// Ошибка датчика давления не останавливает ГВС,
// но переводит подсистему в режим предупреждения (degraded mode).
IF fbPressValidator.VO_Error THEN
    GVL_STATE.G_DHW_Sensor_Fault := TRUE;
    GVL_STATE.G_DHW_Subsystem_Degraded := TRUE;
    VO_Status.Warning := TRUE;
    VO_Status.Error := FALSE;
    VO_Status.Error_ID := TO_WORD(GVL_CONFIG.ERR_DHW_PRESSURE_SENSOR_FAULT);
END_IF;

// 2. Логика поддержания температуры воды в бойлере (Нагрев)
// На этом этапе FB уже выполняется только на активном ПЛК.
    
// Термическая дезинфекция (Легионелла)
IF VI_Config.Anti_Legionella_Enabled
   AND (VI_Current_Day_Of_Week = VI_Config.Anti_Legionella_Day)
   AND (L_Current_TOD >= TOD#02:00)
   AND (L_Current_TOD <= TOD#04:00)
   AND NOT L_Legionella_Done_Today THEN
    L_Legionella_Active := TRUE;
ELSE
    L_Legionella_Active := FALSE;
END_IF;

L_Legionella_Timer(IN := L_Legionella_Active AND VO_Status.Temp >= 70.0, PT := T#30m, VI_System_Time_MS := VI_System_Time_MS);
IF L_Legionella_Timer.Q THEN
    L_Legionella_Active := FALSE; // Дезинфекция завершена
    L_Legionella_Done_Today := TRUE; // Повторно в те же сутки не запускать
END_IF;

// Двухпозиционное регулирование с гистерезисом
IF L_Legionella_Active THEN
    IF VO_Status.Temp < 70.0 THEN
        VO_Heating_Pump := TRUE;
    ELSIF VO_Status.Temp > 72.0 THEN
        VO_Heating_Pump := FALSE;
    END_IF;
ELSE
    IF VO_Status.Temp < (L_Target_Temp_Adjusted - VI_Config.Hysteresis) THEN
        VO_Heating_Pump := TRUE;
    ELSIF VO_Status.Temp > (L_Target_Temp_Adjusted + VI_Config.Hysteresis) THEN
        VO_Heating_Pump := FALSE;
    END_IF;
END_IF;

// 3. Управление циркуляционным насосом ГВС по расписанию
// Рециркуляция обеспечивает мгновенное наличие горячей воды у потребителя
VO_Circ_Pump := SEL(VI_Config.Circulation_Schedule_Enabled AND NOT (VI_Config.Night_Mode_Enabled AND (L_Current_TOD < VI_Config.Circulation_Start OR L_Current_TOD > VI_Config.Circulation_End)), FALSE, TRUE);

// Формирование статусных данных для визуализации.
// К этому моменту статус уже консистентен:
// - Error = критическая ошибка с остановкой ГВС
// - Warning = деградация без остановки
VO_Status.Heating_Pump_On := VO_Heating_Pump;
VO_Status.Circ_Pump_On := VO_Circ_Pump;

// >>> BULK_SYNC_ANCHOR: FB_DHW_Manager <<<
          
END_FUNCTION_BLOCK

FUNCTION_BLOCK FB_Safety_Manager
  VAR_INPUT
    VI_Gas_Alarm : BOOL;
    VI_Leak_Alarm : BOOL;
    VI_Smoke_Alarm : BOOL;
    VI_Reset : BOOL;
  END_VAR
  VAR_OUTPUT
    VO_Gas_Latched : BOOL;
    VO_Leak_Latched : BOOL;
    VO_Smoke_Latched : BOOL;
    VO_Emergency_Stop : BOOL;
  END_VAR
  VAR
    L_Any_Active : BOOL;
  END_VAR

            // Защёлкиваем аварии независимо друг от друга
IF VI_Gas_Alarm THEN
    VO_Gas_Latched := TRUE;
END_IF;

IF VI_Leak_Alarm THEN
    VO_Leak_Latched := TRUE;
END_IF;

IF VI_Smoke_Alarm THEN
    VO_Smoke_Latched := TRUE;
END_IF;

L_Any_Active := VI_Gas_Alarm OR VI_Leak_Alarm OR VI_Smoke_Alarm;

// Ручной сброс допустим только когда все входные аварийные сигналы уже исчезли
IF VI_Reset AND NOT L_Any_Active THEN
    VO_Gas_Latched := FALSE;
    VO_Leak_Latched := FALSE;
    VO_Smoke_Latched := FALSE;
END_IF;

// Агрегированный аварийный стоп = любая защёлкнутая safety-авария
VO_Emergency_Stop := VO_Gas_Latched OR VO_Leak_Latched OR VO_Smoke_Latched;

// >>> BULK_SYNC_ANCHOR: FB_Safety_Manager <<<
          
END_FUNCTION_BLOCK

FUNCTION_BLOCK FB_Calibration_Manager
  VAR_INPUT
    VI_Raw_Value : REAL;
    VI_Type : BYTE;
    VI_Calib_Record : ST_Sensor_Calibration_Record;
    VI_System_Time_MS : UDINT;
    VI_Start_Verification : BOOL;
  END_VAR
  VAR_OUTPUT
    VO_Calibrated_Value : REAL;
    VO_Verification_Active : BOOL;
    VO_Verification_Failed : BOOL;
    VO_Deviation_Percent : REAL;
  END_VAR
  VAR
    L_Verification_Timer : FB_System_Timer;
    L_Initial_Value : REAL;
  END_VAR

            // 1. Расчет калиброванного значения
CASE VI_Type OF
    1: VO_Calibrated_Value := VI_Raw_Value + VI_Calib_Record.offset;
    2, 3: VO_Calibrated_Value := (VI_Raw_Value * VI_Calib_Record.multiplier) + VI_Calib_Record.offset;
END_CASE;

// 2. Верификация через 1 час (ТЗ 9.5)
IF VI_Start_Verification AND NOT VO_Verification_Active THEN
    VO_Verification_Active := TRUE;
    L_Initial_Value := VO_Calibrated_Value;
END_IF;

L_Verification_Timer(IN := VO_Verification_Active, PT := T#1h, VI_System_Time_MS := VI_System_Time_MS);

IF L_Verification_Timer.Q THEN
    VO_Verification_Active := FALSE;
    
    // ТЗ 9.5: Отклонение ≤2.0% (норма) / >5.0% (ошибка)
    IF L_Initial_Value <> 0 THEN
        VO_Deviation_Percent := ABS(VO_Calibrated_Value - L_Initial_Value) / L_Initial_Value * 100.0;
    ELSE
        VO_Deviation_Percent := 0.0;
    END_IF;
    
    VO_Verification_Failed := (VO_Deviation_Percent > 5.0);
END_IF;
          
END_FUNCTION_BLOCK

FUNCTION_BLOCK FB_Persist_Pipeline
  VAR_INPUT
    VI_PersistStruct : ST_Persist;
    VI_System_Time_MS : UDINT;
    VI_IsActivePLC : BOOL;
  END_VAR
  VAR_OUTPUT
    VO_NVRAM_Cmd : BYTE;
    VO_NVRAM_Offset : UDINT;
    VO_NVRAM_Done : BOOL;
    VO_NVRAM_Err : BOOL;
    VO_NVRAM_ErrID : UDINT;
  END_VAR
  VAR_IN_OUT
    VIO_Apply_Settings : BOOL;
    VIO_Persist_Buffer : ARRAY[0..4] OF BYTE;
    VIO_Last_Written_Persist_Buffer : ARRAY[0..4] OF BYTE;
    VIO_Last_Persist_Write_MS : UDINT;
  END_VAR
  VAR
    fbNVRAMManager : FB_NVRAM_Manager;
    L_Persist_Buffer_Changed : BOOL;
  END_VAR

            // === SERIALIZE PERSIST STRUCT → BUFFER ===

// System Mode
VIO_Persist_Buffer[0] := TO_BYTE(TO_INT(VI_PersistStruct.System_Mode));

// Gas
IF VI_PersistStruct.Safety_Gas_Latched THEN
    VIO_Persist_Buffer[1] := BYTE#1;
ELSE
    VIO_Persist_Buffer[1] := BYTE#0;
END_IF;

// Smoke
IF VI_PersistStruct.Safety_Smoke_Latched THEN
    VIO_Persist_Buffer[2] := BYTE#1;
ELSE
    VIO_Persist_Buffer[2] := BYTE#0;
END_IF;

// Leak
IF VI_PersistStruct.Safety_Leak_Latched THEN
    VIO_Persist_Buffer[3] := BYTE#1;
ELSE
    VIO_Persist_Buffer[3] := BYTE#0;
END_IF;

// DHW Pump
IF VI_PersistStruct.DHW_Heating_Pump THEN
    VIO_Persist_Buffer[4] := BYTE#1;
ELSE
    VIO_Persist_Buffer[4] := BYTE#0;
END_IF;

// === END SERIALIZE ===

L_Persist_Buffer_Changed :=
    (VIO_Persist_Buffer[0] <> VIO_Last_Written_Persist_Buffer[0]) OR
    (VIO_Persist_Buffer[1] <> VIO_Last_Written_Persist_Buffer[1]) OR
    (VIO_Persist_Buffer[2] <> VIO_Last_Written_Persist_Buffer[2]) OR
    (VIO_Persist_Buffer[3] <> VIO_Last_Written_Persist_Buffer[3]) OR
    (VIO_Persist_Buffer[4] <> VIO_Last_Written_Persist_Buffer[4]);

VO_NVRAM_Cmd := 0;
VO_NVRAM_Offset := 0;

IF VIO_Apply_Settings THEN
    // explicit config apply requests a controlled write
    // keep flag set until successful write confirmation
    VO_NVRAM_Cmd := 1;

ELSIF L_Persist_Buffer_Changed THEN
    // controlled write: no more often than once per 60 seconds
    IF (VIO_Last_Persist_Write_MS = 0) OR
       ((VI_System_Time_MS - VIO_Last_Persist_Write_MS) >= 60000) THEN
        VO_NVRAM_Cmd := 1;
    END_IF;
END_IF;

fbNVRAMManager(
    VI_Command := VO_NVRAM_Cmd,
    VI_Offset := VO_NVRAM_Offset,
    VI_DataRef := VIO_Persist_Buffer[0],
    VI_DataSize := 5,
    VI_System_Time_MS := VI_System_Time_MS,
    VI_Operator_ID := 'SYSTEM',
    VI_IsActivePLC := VI_IsActivePLC,
    VI_TwoPersonConfirmation := FALSE,
    VO_Done => VO_NVRAM_Done,
    VO_Error => VO_NVRAM_Err,
    VO_ErrorID => VO_NVRAM_ErrID
);

IF (VO_NVRAM_Cmd = 1) AND VO_NVRAM_Done AND NOT VO_NVRAM_Err THEN
    VIO_Last_Written_Persist_Buffer[0] := VIO_Persist_Buffer[0];
    VIO_Last_Written_Persist_Buffer[1] := VIO_Persist_Buffer[1];
    VIO_Last_Written_Persist_Buffer[2] := VIO_Persist_Buffer[2];
    VIO_Last_Written_Persist_Buffer[3] := VIO_Persist_Buffer[3];
    VIO_Last_Written_Persist_Buffer[4] := VIO_Persist_Buffer[4];
    VIO_Last_Persist_Write_MS := VI_System_Time_MS;
    VIO_Apply_Settings := FALSE;
END_IF;
          
END_FUNCTION_BLOCK

FUNCTION_BLOCK FB_Boiler_Cascade_Manager
  VAR_INPUT
    VI_Enable : BOOL;
    VI_System_Time_MS : UDINT;
    VI_Boiler_Stop : BOOL;
    VI_DHW_Heating_Demand : BOOL;
    VI_DHW_Target_Temp : REAL;
    VI_Target_Supply_Temp : REAL;
    VI_Demand_Power : REAL;
    VI_Boiler_Flame_Status : ARRAY[1..GVL_CONSTANTS.C_MAX_BOILERS] OF BOOL;
    VI_Boiler_Error_Status : ARRAY[1..GVL_CONSTANTS.C_MAX_BOILERS] OF BOOL;
    VI_Boiler_OT_Online : ARRAY[1..GVL_CONSTANTS.C_MAX_BOILERS] OF BOOL;
    VI_Boiler_Modulation : ARRAY[1..GVL_CONSTANTS.C_MAX_BOILERS] OF REAL;
  END_VAR
  VAR_OUTPUT
    VO_Boiler_Enable : ARRAY[1..GVL_CONSTANTS.C_MAX_BOILERS] OF BOOL;
    VO_Boiler_Setpoint : ARRAY[1..GVL_CONSTANTS.C_MAX_BOILERS] OF REAL;
    VO_Lead_Boiler : BYTE;
  END_VAR
  VAR
    L_i : INT;
    L_Lead_Boiler : BYTE := 1;
    L_Last_Rotation_MS : UDINT := 0;
    L_Rotation_Initialized : BOOL := FALSE;
    L_Rotation_Period_MS : UDINT := 604800000;
    L_Lead_Available : BOOL;
    L_Reserve_Available : BOOL;
    L_Reserve_Boiler : BYTE;
    L_Start_Reserve : BOOL;
    L_Target_Setpoint : REAL;
    L_Flame_Miss_Timer : ARRAY[1..GVL_CONSTANTS.C_MAX_BOILERS] OF TON;
  END_VAR

            // Сброс выходов по умолчанию
FOR L_i := 1 TO GVL_CONSTANTS.C_MAX_BOILERS DO
    VO_Boiler_Enable[L_i] := FALSE;
    VO_Boiler_Setpoint[L_i] := 0.0;
END_FOR;

// Инициализация ротации
IF NOT L_Rotation_Initialized THEN
    L_Last_Rotation_MS := VI_System_Time_MS;
    L_Rotation_Initialized := TRUE;
END_IF;

// Принудительная остановка
IF VI_Boiler_Stop THEN
    VO_Lead_Boiler := L_Lead_Boiler;
    RETURN;
END_IF;

// Ротация строго каждые 168 часов
IF (VI_System_Time_MS - L_Last_Rotation_MS) >= L_Rotation_Period_MS THEN
    IF GVL_CONSTANTS.C_MAX_BOILERS > 1 THEN
        L_Lead_Boiler := 3 - L_Lead_Boiler;
    END_IF;
    L_Last_Rotation_MS := VI_System_Time_MS;
END_IF;

L_Reserve_Boiler := SEL(L_Lead_Boiler = 1, 1, 2);

L_Lead_Available :=
    VI_Boiler_OT_Online[L_Lead_Boiler] AND
    NOT VI_Boiler_Error_Status[L_Lead_Boiler];

L_Reserve_Available :=
    (GVL_CONSTANTS.C_MAX_BOILERS > 1) AND
    VI_Boiler_OT_Online[L_Reserve_Boiler] AND
    NOT VI_Boiler_Error_Status[L_Reserve_Boiler];

// Контроль "команда есть, пламени нет" для ведущего котла
L_Flame_Miss_Timer[L_Lead_Boiler](
    IN := VI_Enable AND L_Lead_Available AND NOT VI_DHW_Heating_Demand AND NOT VI_Boiler_Flame_Status[L_Lead_Boiler],
    PT := T#120s
);

IF L_Flame_Miss_Timer[L_Lead_Boiler].Q AND L_Reserve_Available THEN
    L_Lead_Boiler := L_Reserve_Boiler;
    L_Last_Rotation_MS := VI_System_Time_MS;
    L_Lead_Available :=
        VI_Boiler_OT_Online[L_Lead_Boiler] AND
        NOT VI_Boiler_Error_Status[L_Lead_Boiler];
    L_Reserve_Boiler := SEL(L_Lead_Boiler = 1, 1, 2);
    L_Reserve_Available :=
        (GVL_CONSTANTS.C_MAX_BOILERS > 1) AND
        VI_Boiler_OT_Online[L_Reserve_Boiler] AND
        NOT VI_Boiler_Error_Status[L_Reserve_Boiler];
END_IF;

// Нет запроса тепла
IF NOT VI_Enable THEN
    VO_Lead_Boiler := L_Lead_Boiler;
    RETURN;
END_IF;

// Целевая уставка
IF VI_DHW_Heating_Demand THEN
    L_Target_Setpoint := LIMIT(20.0, VI_DHW_Target_Temp + 15.0, 85.0);
ELSE
    L_Target_Setpoint := LIMIT(20.0, VI_Target_Supply_Temp + 5.0, 80.0);
END_IF;

// Выбор ведущего по доступности
IF NOT L_Lead_Available AND L_Reserve_Available THEN
    L_Lead_Boiler := L_Reserve_Boiler;
    L_Lead_Available := TRUE;
    L_Reserve_Boiler := SEL(L_Lead_Boiler = 1, 1, 2);
    L_Reserve_Available :=
        (GVL_CONSTANTS.C_MAX_BOILERS > 1) AND
        VI_Boiler_OT_Online[L_Reserve_Boiler] AND
        NOT VI_Boiler_Error_Status[L_Reserve_Boiler];
END_IF;

// Основной котёл
IF L_Lead_Available THEN
    VO_Boiler_Enable[L_Lead_Boiler] := TRUE;
    VO_Boiler_Setpoint[L_Lead_Boiler] := L_Target_Setpoint;
END_IF;

// Резервный котёл: >80% или отказ основного
L_Start_Reserve :=
    L_Reserve_Available AND
    (
        (VI_Demand_Power > 80.0) OR
        (NOT L_Lead_Available)
    );

IF L_Start_Reserve THEN
    VO_Boiler_Enable[L_Reserve_Boiler] := TRUE;
    VO_Boiler_Setpoint[L_Reserve_Boiler] := L_Target_Setpoint;
END_IF;

VO_Lead_Boiler := L_Lead_Boiler;
          
END_FUNCTION_BLOCK

FUNCTION_BLOCK FB_Watchdog
  VAR_INPUT
    VI_System_Time_MS : UDINT;
    VI_Timeout_MS : UDINT := 2000;
  END_VAR
  VAR_OUTPUT
    VO_Alive : BOOL;
    VO_Watchdog_Fault : BOOL;
    VO_Cycle_DT_MS : UDINT;
  END_VAR
  VAR
    L_Initialized : BOOL := FALSE;
    L_Last_Call_MS : UDINT := 0;
    L_DT_MS : UDINT := 0;
  END_VAR

            IF NOT L_Initialized THEN
    L_Initialized := TRUE;
    L_Last_Call_MS := VI_System_Time_MS;
    VO_Cycle_DT_MS := 0;
    VO_Watchdog_Fault := FALSE;
    VO_Alive := TRUE;
    RETURN;
END_IF;

// Measure real time gap between successive calls
L_DT_MS := (SEL(VI_System_Time_MS >= L_Last_Call_MS, VI_System_Time_MS - L_Last_Call_MS, (4294967295 - L_Last_Call_MS) + VI_System_Time_MS + 1));
VO_Cycle_DT_MS := L_DT_MS;

// Fault if the task/cycle resumed after an abnormal pause
VO_Watchdog_Fault := (L_DT_MS > VI_Timeout_MS);
VO_Alive := NOT VO_Watchdog_Fault;

// Store current timestamp for next cycle
L_Last_Call_MS := VI_System_Time_MS;
// >>> BULK_SYNC_ANCHOR: FB_Watchdog <<<
          
END_FUNCTION_BLOCK

FUNCTION_BLOCK FB_System_Health_Orchestrator
  VAR_OUTPUT
    VO_First_Fault_Active : BOOL;
    VO_First_Fault_Type : INT;
    VO_First_Fault_Source : INT;
    VO_System_Severity : E_System_Severity;
    VO_Root_Cause : E_System_Root_Cause;
    VO_Watchdog_Fault : BOOL;
  END_VAR
  VAR
    fbSafety : FB_Safety_Manager;
    fbWatchdog : FB_Watchdog;
    fbSystemHealth : FB_System_Health;
    fbStateManager : FB_State_Manager;
    fbHMIInterface : FB_HMI_Interface;
    fbFaultLogger : FB_Fault_Logger;
  END_VAR

            // ==============================================================================
// System health orchestrator helper
//
// Internal helper for PRG_System.
// Owns safety latch update, watchdog, system health aggregation,
// system mode calculation, HMI/fault publication, diagnostic exports,
// and human-readable mode/cause text projection.
// ==============================================================================



fbSafety(
    VI_Gas_Alarm := GVL_STATE.G_Safety_Gas_Alarm,
    VI_Leak_Alarm := GVL_STATE.G_Safety_Leak_Alarm,
    VI_Smoke_Alarm := GVL_STATE.G_Safety_Smoke_Alarm,
    VI_Reset := GVL_COMMAND.G_Reset_Errors,
    VO_Gas_Latched => GVL_STATE.G_Safety_Gas_Latched,
    VO_Leak_Latched => GVL_STATE.G_Safety_Leak_Latched,
    VO_Smoke_Latched => GVL_STATE.G_Safety_Smoke_Latched,
    VO_Emergency_Stop => GVL_STATE.G_Safety_Emergency_Stop
);

GVL_STATE.G_Freeze_Hardware_Degraded := GVL_STATUS.G_Diagnostics.Backup_Pump_Fault OR GVL_STATUS.G_Diagnostics.Electric_Heater_Fault;
GVL_STATE.G_Freeze_Hardware_Failed := GVL_STATUS.G_Diagnostics.Backup_Pump_Fault AND GVL_STATUS.G_Diagnostics.Electric_Heater_Fault;

fbWatchdog(
    VI_System_Time_MS := GVL_STATUS.G_System_Time_MS
);

fbSystemHealth(
    VI_Smoke_Detected := GVL_HEALTH_BRIDGE.G_Smoke_Detected OR GVL_STATE.G_Safety_Smoke_Latched,
    VI_Gas_Detected := GVL_HEALTH_BRIDGE.G_Gas_Detected OR GVL_STATE.G_Safety_Gas_Latched,
    VI_CO_Warning_Level := GVL_HEALTH_BRIDGE.G_CO_Warning_Level,
    VI_CO_Alarm_Level := GVL_HEALTH_BRIDGE.G_CO_Alarm_Level,
    VI_Leak_Detected := GVL_HEALTH_BRIDGE.G_Leak_Detected OR GVL_STATE.G_Safety_Leak_Latched,
    VI_Sensor_Fault := GVL_STATE.G_Heating_Sensor_Fault OR GVL_STATE.G_DHW_Sensor_Fault OR GVL_STATUS.G_Diagnostics.Manifold_Pressure_Fault_Active OR GVL_STATUS.G_Diagnostics.Manifold_Current_Fault_Active OR GVL_STATUS.G_Diagnostics.Manifold_Return_Temp_Fault_Active,
    VI_IO_Offline := GVL_STATE.G_Heating_IO_Fault OR GVL_STATE.G_DHW_IO_Fault OR GVL_STATE.G_Ventilation_IO_Fault OR GVL_STATE.G_Lighting_IO_Fault,
    VI_Comm_Fault := GVL_STATE.G_Access_Comm_Fault,
    VI_Watchdog_Fault := fbWatchdog.VO_Watchdog_Fault,
    VI_Subsystem_Fault := GVL_STATE.G_Heating_Subsystem_Degraded OR GVL_STATE.G_DHW_Subsystem_Degraded OR GVL_STATE.G_Ventilation_Subsystem_Degraded OR GVL_STATUS.G_Diagnostics.Manifold_Pressure_Fault_Active OR GVL_STATUS.G_Diagnostics.Manifold_Current_Fault_Active OR GVL_STATUS.G_Diagnostics.Manifold_Return_Temp_Fault_Active
);

fbStateManager(
    VI_System_Severity := fbSystemHealth.VO_System_Severity,
    VI_Root_Cause := fbSystemHealth.VO_Root_Cause,
    VI_Freeze_Risk := GVL_STATE.G_Safety_Freeze_Risk
);

fbHMIInterface(
    VI_Severity := fbSystemHealth.VO_System_Severity,
    VI_RootCause := fbSystemHealth.VO_Root_Cause,
    VI_Status_Msg := fbStateManager.VO_Status_Msg
);

fbFaultLogger(
    VI_Severity := fbSystemHealth.VO_System_Severity,
    VI_RootCause := fbSystemHealth.VO_Root_Cause,
    VI_Time_MS := GVL_STATUS.G_System_Time_MS
);

GVL_STATUS.G_System_Mode_Msg := fbStateManager.VO_Status_Msg;

GVL_STATUS.G_Diagnostics.Sensor_Fault :=
    GVL_STATE.G_Heating_Sensor_Fault OR
    GVL_STATE.G_DHW_Sensor_Fault OR
    GVL_STATUS.G_Diagnostics.Manifold_Pressure_Fault_Active OR
    GVL_STATUS.G_Diagnostics.Manifold_Current_Fault_Active OR
    GVL_STATUS.G_Diagnostics.Manifold_Return_Temp_Fault_Active;

GVL_STATUS.G_Diagnostics.IO_Offline :=
    GVL_STATE.G_Heating_IO_Fault OR
    GVL_STATE.G_DHW_IO_Fault OR
    GVL_STATE.G_Ventilation_IO_Fault OR
    GVL_STATE.G_Lighting_IO_Fault;

GVL_STATUS.G_Diagnostics.Subsystem_Degraded :=
    GVL_STATE.G_Heating_Subsystem_Degraded OR
    GVL_STATE.G_DHW_Subsystem_Degraded OR
    GVL_STATE.G_Ventilation_Subsystem_Degraded OR
    GVL_STATUS.G_Diagnostics.Manifold_Pressure_Fault_Active OR
    GVL_STATUS.G_Diagnostics.Manifold_Current_Fault_Active OR
    GVL_STATUS.G_Diagnostics.Manifold_Return_Temp_Fault_Active;

GVL_GATEWAY.G_Gateway_HMI_Status_Message := fbHMIInterface.VO_HMI_Status_Text;
IF fbFaultLogger.VO_Last_Event_Text <> '' THEN
    GVL_HEALTH_BRIDGE.G_Last_Fault_Event_Text := fbFaultLogger.VO_Last_Event_Text;
END_IF;

GVL_STATE.G_System_Mode := fbStateManager.VO_System_Mode;

CASE GVL_STATE.G_System_Mode OF
    E_System_Operating_Mode.MODE_SAFE_STOP:
        GVL_STATE.G_System_Mode_Text := 'SAFE_STOP';

    E_System_Operating_Mode.MODE_FREEZE_PROTECTION:
        GVL_STATE.G_System_Mode_Text := 'FREEZE_PROTECTION';

    E_System_Operating_Mode.MODE_DEGRADED:
        GVL_STATE.G_System_Mode_Text := 'DEGRADED';

    ELSE
        GVL_STATE.G_System_Mode_Text := 'NORMAL';
END_CASE;

CASE fbSystemHealth.VO_Root_Cause OF
    E_System_Root_Cause.ROOT_FIRE:
        GVL_STATUS.G_System_Mode_Cause := 'Пожар/дым';
    E_System_Root_Cause.ROOT_GAS_LEAK:
        GVL_STATUS.G_System_Mode_Cause := 'Утечка газа';
    E_System_Root_Cause.ROOT_CO_CRITICAL:
        GVL_STATUS.G_System_Mode_Cause := 'Критический CO';
    E_System_Root_Cause.ROOT_CO_WARNING:
        GVL_STATUS.G_System_Mode_Cause := 'Повышенный CO';
    E_System_Root_Cause.ROOT_WATER_LEAK:
        GVL_STATUS.G_System_Mode_Cause := 'Протечка воды';
    E_System_Root_Cause.ROOT_WATCHDOG_FAULT:
        GVL_STATUS.G_System_Mode_Cause := 'Ошибка watchdog';
    E_System_Root_Cause.ROOT_IO_OFFLINE:
        GVL_STATUS.G_System_Mode_Cause := 'Недоступен модуль IO';
    E_System_Root_Cause.ROOT_COMM_FAULT:
        GVL_STATUS.G_System_Mode_Cause := 'Ошибка связи';
    E_System_Root_Cause.ROOT_SENSOR_FAULT:
        GVL_STATUS.G_System_Mode_Cause := 'Ошибка датчика';
    E_System_Root_Cause.ROOT_SUBSYSTEM_FAULT:
        GVL_STATUS.G_System_Mode_Cause := 'Ошибка подсистемы';
    ELSE
        GVL_STATUS.G_System_Mode_Cause := 'Аварийные режимы отсутствуют';
END_CASE;

VO_First_Fault_Active := fbSystemHealth.VO_First_Fault_Active;
VO_First_Fault_Type := fbSystemHealth.VO_First_Fault_Type;
VO_First_Fault_Source := fbSystemHealth.VO_First_Fault_Source;
VO_System_Severity := fbSystemHealth.VO_System_Severity;
VO_Root_Cause := fbSystemHealth.VO_Root_Cause;
VO_Watchdog_Fault := fbWatchdog.VO_Watchdog_Fault;

GVL_STATUS.G_System_Mode_Msg := fbStateManager.VO_Status_Msg;

// >>> BULK_SYNC_ANCHOR: FB_System_Health_Orchestrator <<<
          
END_FUNCTION_BLOCK

FUNCTION_BLOCK FB_Diagnostics_Event_Manager
  VAR_INPUT
    VI_Code : UDINT;
    VI_Severity : INT;
    VI_Active : BOOL;
    VI_Timestamp : UDINT;
    VI_Source : INT;
  END_VAR
  VAR_IN_OUT
    VIO_Events : ARRAY[1..50] OF ST_Diagnostic_Event;
    VIO_Count : INT;
  END_VAR
  VAR
    L_i : INT;
    L_Found_Index : INT;
    L_Was_Active : BOOL;
  END_VAR

            L_Found_Index := 0;
L_Was_Active := FALSE;

FOR L_i := 1 TO VIO_Count DO
    IF (VIO_Events[L_i].Code = VI_Code) AND (VIO_Events[L_i].Source = VI_Source) THEN
        L_Found_Index := L_i;
        L_Was_Active := VIO_Events[L_i].Active;
    END_IF;
END_FOR;

IF VI_Active THEN
    IF L_Found_Index = 0 THEN
        IF VIO_Count < 50 THEN
            VIO_Count := VIO_Count + 1;
            VIO_Events[VIO_Count].Code := VI_Code;
            VIO_Events[VIO_Count].Severity := VI_Severity;
            VIO_Events[VIO_Count].Active := TRUE;
            VIO_Events[VIO_Count].Timestamp := VI_Timestamp;
            VIO_Events[VIO_Count].Source := VI_Source;
        END_IF;
    ELSE
        VIO_Events[L_Found_Index].Severity := VI_Severity;
        IF NOT L_Was_Active THEN
            VIO_Events[L_Found_Index].Timestamp := VI_Timestamp;
        END_IF;
        VIO_Events[L_Found_Index].Active := TRUE;
    END_IF;
ELSE
    IF L_Found_Index > 0 THEN
        VIO_Events[L_Found_Index].Active := FALSE;
    END_IF;
END_IF;
          
END_FUNCTION_BLOCK

PROGRAM PRG_Command_Arbitration
  VAR
    L_i : INT;
  END_VAR

            // Reset shadow operational commands before each arbitration cycle
GVL_COMMAND_SHADOW.G_Gas_Valve_Close := FALSE;
GVL_COMMAND_SHADOW.G_Boiler_Stop := FALSE;
GVL_COMMAND_SHADOW.G_Supply_100_Req := FALSE;
GVL_COMMAND_SHADOW.G_Supply_80_Req := FALSE;
GVL_COMMAND_SHADOW.G_Vent_PV3_Boost := FALSE;
GVL_COMMAND_SHADOW.G_Exhaust_100_Req := FALSE;
GVL_COMMAND_SHADOW.G_Vent_Stop := FALSE;

GVL_COMMAND_SHADOW.G_Close_Valve_35 := FALSE;
GVL_COMMAND_SHADOW.G_Close_Valve_36 := FALSE;

GVL_COMMAND_SHADOW.G_Lock_1_Open := FALSE;
GVL_COMMAND_SHADOW.G_Lock_1_Close := FALSE;
GVL_COMMAND_SHADOW.G_Lock_2_Open := FALSE;
GVL_COMMAND_SHADOW.G_Lock_2_Close := FALSE;
GVL_COMMAND_SHADOW.G_Gate_Open := FALSE;
GVL_COMMAND_SHADOW.G_Wicket_Open := FALSE;

// User intent pass-through into the shadow operational layer
GVL_COMMAND_SHADOW.G_Gate_Open := GVL_INTENT_USER.I_Gate_Open_Request;
GVL_COMMAND_SHADOW.G_Wicket_Open := GVL_INTENT_USER.I_Wicket_Open_Request;
GVL_COMMAND_SHADOW.G_Lock_1_Open := GVL_INTENT_USER.I_Lock_1_Open_Request;
GVL_COMMAND_SHADOW.G_Lock_1_Close := GVL_INTENT_USER.I_Lock_1_Close_Request;
GVL_COMMAND_SHADOW.G_Lock_2_Open := GVL_INTENT_USER.I_Lock_2_Open_Request;
GVL_COMMAND_SHADOW.G_Lock_2_Close := GVL_INTENT_USER.I_Lock_2_Close_Request;

// Safety and system arbitration into the shadow operational layer
IF GVL_INTENT_SAFETY.I_Fire_Alarm_Active THEN
    GVL_COMMAND_SHADOW.G_Boiler_Stop := TRUE;
    GVL_COMMAND_SHADOW.G_Vent_Stop := TRUE;
    GVL_COMMAND_SHADOW.G_Lock_1_Open := TRUE;
    GVL_COMMAND_SHADOW.G_Lock_2_Open := TRUE;
END_IF;

IF GVL_INTENT_SAFETY.I_Gas_Close_Required THEN
    GVL_COMMAND_SHADOW.G_Gas_Valve_Close := TRUE;
    GVL_COMMAND_SHADOW.G_Boiler_Stop := TRUE;
END_IF;

IF GVL_INTENT_SAFETY.I_Vent_Force_PV3_Boost THEN
    GVL_COMMAND_SHADOW.G_Vent_PV3_Boost := TRUE;
END_IF;

IF GVL_INTENT_SAFETY.I_Vent_Force_Supply_100 THEN
    GVL_COMMAND_SHADOW.G_Supply_100_Req := TRUE;
END_IF;

IF GVL_INTENT_SAFETY.I_Vent_Force_Supply_80 THEN
    GVL_COMMAND_SHADOW.G_Supply_80_Req := TRUE;
END_IF;

IF GVL_INTENT_SAFETY.I_Vent_Stop_Required THEN
    GVL_COMMAND_SHADOW.G_Vent_Stop := TRUE;
END_IF;

IF GVL_INTENT_SYSTEM.I_Mode_Degraded_Active THEN
    GVL_COMMAND_SHADOW.G_Supply_80_Req := TRUE;
END_IF;

IF GVL_INTENT_SAFETY.I_Water_Main_Close_Required THEN
    GVL_COMMAND_SHADOW.G_Close_Valve_35 := TRUE;
    GVL_COMMAND_SHADOW.G_Close_Valve_36 := TRUE;
END_IF;

FOR L_i := 1 TO 32 DO
    IF GVL_INTENT_SAFETY.I_Water_Zone_Close_Required[L_i] THEN
        ;
    END_IF;
END_FOR;
          
END_PROGRAM

PROGRAM PRG_PLC_A

            // Вызов основной программы
PRG_System();
// >>> BULK_SYNC_ANCHOR: PRG_PLC_A <<<
          
END_PROGRAM

PROGRAM PRG_Policy

            // ============================================================
// SCENARIO POLICY OWNER
// ============================================================

// 1. Base priority resolution
IF GVL_STATE.G_System_Mode = E_System_Operating_Mode.MODE_SAFE_STOP THEN
    GVL_POLICY.G_Scenario_Intent := E_SCENARIO_TYPE.SCENARIO_NONE;
    GVL_POLICY.G_Scenario_Source := SRC_SAFETY;

ELSIF GVL_POLICY.G_Scenario_Request_Operator <> E_SCENARIO_TYPE.SCENARIO_NONE THEN
    GVL_POLICY.G_Scenario_Intent := GVL_POLICY.G_Scenario_Request_Operator;
    GVL_POLICY.G_Scenario_Source := SRC_OPERATOR;

ELSIF GVL_POLICY.G_Scenario_Request_Gateway <> E_SCENARIO_TYPE.SCENARIO_NONE THEN
    GVL_POLICY.G_Scenario_Intent := GVL_POLICY.G_Scenario_Request_Gateway;
    GVL_POLICY.G_Scenario_Source := SRC_GATEWAY;

ELSIF GVL_POLICY.G_Scenario_Request_Rule <> E_SCENARIO_TYPE.SCENARIO_NONE THEN
    GVL_POLICY.G_Scenario_Intent := GVL_POLICY.G_Scenario_Request_Rule;
    GVL_POLICY.G_Scenario_Source := SRC_RULE;

ELSE
    GVL_POLICY.G_Scenario_Intent := GVL_STATUS.G_Current_Scenario;
    GVL_POLICY.G_Scenario_Source := SRC_NONE;
END_IF;

// 2. Fail-safe clamp
CASE GVL_STATE.G_System_Mode OF
    E_System_Operating_Mode.MODE_SAFE_STOP:
        GVL_POLICY.G_Scenario_Intent := E_SCENARIO_TYPE.SCENARIO_NONE;
        GVL_POLICY.G_Scenario_Source := SRC_SAFETY;

    E_System_Operating_Mode.MODE_FREEZE_PROTECTION:
        GVL_POLICY.G_Scenario_Intent := E_SCENARIO_TYPE.SCENARIO_NONE;
        GVL_POLICY.G_Scenario_Source := SRC_POLICY;

    E_System_Operating_Mode.MODE_DEGRADED:
        CASE GVL_POLICY.G_Scenario_Intent OF
            E_SCENARIO_TYPE.SCENARIO_NONE,
            E_SCENARIO_TYPE.SCENARIO_PRESENCE,
            E_SCENARIO_TYPE.SCENARIO_AWAY,
            E_SCENARIO_TYPE.SCENARIO_SLEEP:
                ;
        ELSE
            GVL_POLICY.G_Scenario_Intent := E_SCENARIO_TYPE.SCENARIO_NONE;
            GVL_POLICY.G_Scenario_Source := SRC_POLICY;
        END_CASE;
END_CASE;

// 3. Context automation
IF GVL_STATE.G_System_Mode = E_System_Operating_Mode.MODE_NORMAL THEN
    IF GVL_ALARM.G_Security_Armed AND
       (GVL_POLICY.G_Scenario_Request_Operator = E_SCENARIO_TYPE.SCENARIO_NONE) AND
       (GVL_POLICY.G_Scenario_Request_Gateway = E_SCENARIO_TYPE.SCENARIO_NONE) AND
       (GVL_POLICY.G_Scenario_Request_Rule = E_SCENARIO_TYPE.SCENARIO_NONE) AND
       (GVL_POLICY.G_Scenario_Intent <> E_SCENARIO_TYPE.SCENARIO_AWAY) THEN
        GVL_POLICY.G_Scenario_Intent := E_SCENARIO_TYPE.SCENARIO_AWAY;
        GVL_POLICY.G_Scenario_Source := SRC_POLICY;
    END_IF;
END_IF;

// 4. Degraded adaptation
IF GVL_STATE.G_System_Mode = E_System_Operating_Mode.MODE_DEGRADED THEN
    IF (GVL_POLICY.G_Scenario_Request_Operator = E_SCENARIO_TYPE.SCENARIO_NONE) AND
       (GVL_POLICY.G_Scenario_Request_Gateway = E_SCENARIO_TYPE.SCENARIO_NONE) AND
       (GVL_POLICY.G_Scenario_Request_Rule = E_SCENARIO_TYPE.SCENARIO_NONE) THEN

        IF GVL_ALARM.G_Security_Armed THEN
            GVL_POLICY.G_Scenario_Intent := E_SCENARIO_TYPE.SCENARIO_AWAY;
            GVL_POLICY.G_Scenario_Source := SRC_POLICY;

        ELSIF GVL_POLICY.G_Scenario_Intent = E_SCENARIO_TYPE.SCENARIO_PRESENCE THEN
            GVL_POLICY.G_Scenario_Intent := E_SCENARIO_TYPE.SCENARIO_SLEEP;
            GVL_POLICY.G_Scenario_Source := SRC_POLICY;
        END_IF;
    END_IF;
END_IF;

// 5. Heating bridge
GVL_STATE.G_Preheat_Request := GVL_POLICY.G_Rule_Preheat_Request;
GVL_STATE.G_Freeze_Request :=
    (GVL_STATE.G_System_Mode = E_System_Operating_Mode.MODE_FREEZE_PROTECTION);
          
END_PROGRAM

PROGRAM PRG_Safety
  VAR
    fbWaterLeakageManager : FB_Water_Leakage_Manager;
    fbGasSmokeManager : FB_Gas_Smoke_Manager;
    fbSafetyWorkflow : FB_Safety_Workflow_Manager;
    fbOwnership : FB_Ownership_Watchdog;
    L_i : INT;
  END_VAR

            // ========================================
// SAFETY_INTENT_RESET_INIT
// ========================================
GVL_INTENT_SAFETY.I_Source_Valid := TRUE;
GVL_INTENT_SAFETY.I_Last_Update_MS := GVL_STATUS.G_System_Time_MS;
GVL_INTENT_SAFETY.I_Fire_Alarm_Active := FALSE;
GVL_INTENT_SAFETY.I_Gas_Alarm_Active := FALSE;
GVL_INTENT_SAFETY.I_Leak_Alarm_Active := FALSE;
GVL_INTENT_SAFETY.I_CO_Warning_Active := FALSE;
GVL_INTENT_SAFETY.I_System_Safe_Stop_Required := FALSE;
GVL_INTENT_SAFETY.I_Freeze_Protection_Required := FALSE;
GVL_INTENT_SAFETY.I_Evacuation_Mode_Active := FALSE;
GVL_INTENT_SAFETY.I_Gas_Close_Required := FALSE;
GVL_INTENT_SAFETY.I_Boiler_Stop_Required := FALSE;
GVL_INTENT_SAFETY.I_Vent_Stop_Required := FALSE;
GVL_INTENT_SAFETY.I_Vent_Force_PV3_Boost := FALSE;
GVL_INTENT_SAFETY.I_Vent_Force_Supply_100 := FALSE;
GVL_INTENT_SAFETY.I_Vent_Force_Supply_80 := FALSE;
GVL_INTENT_SAFETY.I_Vent_Force_Exhaust_100 := FALSE;
GVL_INTENT_SAFETY.I_Water_Main_Close_Required := FALSE;
GVL_INTENT_SAFETY.I_Water_Selective_Recovery_Allowed := FALSE;
GVL_INTENT_SAFETY.I_Water_Recovery_Target_Zone := 0;
GVL_INTENT_SAFETY.I_Lock_1_Force_Open := FALSE;
GVL_INTENT_SAFETY.I_Lock_1_Force_Close_Block := FALSE;
GVL_INTENT_SAFETY.I_Lock_2_Force_Open := FALSE;
GVL_INTENT_SAFETY.I_Lock_2_Force_Close_Block := FALSE;

// ========================================
// SAFETY_WORKFLOW_FB
// ========================================
fbSafetyWorkflow(
    VI_System_Time_MS := GVL_STATUS.G_System_Time_MS,
    VI_Water_Selective_Recover := GVL_INTENT_USER.I_Water_Selective_Recover,
    VI_Gas_Selective_Recover := GVL_INTENT_USER.I_Gas_Selective_Recover,
    VI_Water_Valve_Test_Open := GVL_INTENT_USER.I_Water_Valve_Test_Open,
    VI_Water_Valve_Test_Close := GVL_INTENT_USER.I_Water_Valve_Test_Close,
    VI_Water_Valve_Test_Confirm := GVL_INTENT_USER.I_Water_Valve_Test_Confirm,
    VI_Gas_Valve_Test_Open := GVL_INTENT_USER.I_Gas_Valve_Test_Open,
    VI_Gas_Valve_Test_Close := GVL_INTENT_USER.I_Gas_Valve_Test_Close,
    VI_Gas_Valve_Test_Confirm := GVL_INTENT_USER.I_Gas_Valve_Test_Confirm
);

IF fbSafetyWorkflow.VO_Water_Test_Timeout_Close_Required THEN
    GVL_INTENT_SAFETY.I_Water_Main_Close_Required := TRUE;
END_IF;

IF fbSafetyWorkflow.VO_Gas_Test_Timeout_Close_Required THEN
    GVL_INTENT_SAFETY.I_Gas_Close_Required := TRUE;
END_IF;

// ========================================
// SAFETY_DETECTORS_AND_HEALTH_PROJECTION
// ========================================
fbWaterLeakageManager(
    VI_System_Time_MS := GVL_STATUS.G_System_Time_MS,
    VI_IsActivePLC := GVL_STATUS.G_Is_Active_PLC,
    VI_Sensors := GVL_STATE.G_Water_Sensors,
    VI_Config := GVL_CONFIG.G_HMI_Flood_Config,
    VO_Status_Msg => GVL_STATUS.G_Flood_Status_Msg,
    VO_Leak_Detected => GVL_HEALTH_BRIDGE.G_Leak_Detected,
    VO_Leak_Warning_Level => GVL_HEALTH_BRIDGE.G_Leak_Warning_Level
);
GVL_INTENT_SAFETY.I_Leak_Alarm_Active := GVL_HEALTH_BRIDGE.G_Leak_Detected;

fbGasSmokeManager(
    VI_System_Time_MS := GVL_STATUS.G_System_Time_MS,
    VI_IsActivePLC := GVL_STATUS.G_Is_Active_PLC,
    VI_Methane_LEL := GVL_Safety_Selector.G_Methane_Effective_Array,
    VI_CO_PPM := GVL_Safety_Selector.G_CO_Effective_Array,
    VI_Smoke_Sensors := GVL_Safety_Selector.G_Smoke_Effective_Array,
    VI_Mute_Request := GVL_CONFIG.G_HMI_Mute_Alarm,
    VO_Smoke_Detected => GVL_HEALTH_BRIDGE.G_Smoke_Detected,
    VO_Gas_Detected => GVL_HEALTH_BRIDGE.G_Gas_Detected,
    VO_CO_Warning_Level => GVL_HEALTH_BRIDGE.G_CO_Warning_Level,
    VO_CO_Alarm_Level => GVL_HEALTH_BRIDGE.G_CO_Alarm_Level,
    VO_Status_Msg => GVL_STATUS.G_Gas_Status_Msg
);
GVL_INTENT_SAFETY.I_Fire_Alarm_Active := GVL_HEALTH_BRIDGE.G_Smoke_Detected;
GVL_INTENT_SAFETY.I_Gas_Alarm_Active := GVL_HEALTH_BRIDGE.G_Gas_Detected OR GVL_HEALTH_BRIDGE.G_CO_Alarm_Level;
GVL_INTENT_SAFETY.I_CO_Warning_Active := GVL_HEALTH_BRIDGE.G_CO_Warning_Level;

// ========================================
// OWNERSHIP WATCHDOG
// ========================================
fbOwnership(
    VI_Gas_Level := GVL_STATE.G_Methane_Sensors[1],
    VI_Gas_Alarm := GVL_STATE.G_Safety_Gas_Alarm,
    VI_Leak_Alarm := GVL_STATE.G_Safety_Leak_Alarm,
    VI_Smoke_Alarm := GVL_STATE.G_Safety_Smoke_Alarm
);

IF fbOwnership.VO_Ownership_Violation THEN
    GVL_TEST.G_Ownership_Violation := TRUE;
END_IF;

// ========================================
// SAFETY_CORE_HAZARD_INTERLOCK_PROJECTION
// ========================================
IF GVL_STATE.G_Safety_Smoke_Latched THEN
    GVL_INTENT_SAFETY.I_System_Safe_Stop_Required := TRUE;
    GVL_INTENT_SAFETY.I_Evacuation_Mode_Active := TRUE;
    GVL_INTENT_SAFETY.I_Boiler_Stop_Required := TRUE;
    GVL_INTENT_SAFETY.I_Vent_Stop_Required := TRUE;
    GVL_INTENT_SAFETY.I_Lock_1_Force_Open := TRUE;
    GVL_INTENT_SAFETY.I_Lock_1_Force_Close_Block := TRUE;
    GVL_INTENT_SAFETY.I_Lock_2_Force_Open := TRUE;
    GVL_INTENT_SAFETY.I_Lock_2_Force_Close_Block := TRUE;
END_IF;

IF GVL_STATE.G_Safety_Gas_Latched THEN
    GVL_INTENT_SAFETY.I_System_Safe_Stop_Required := TRUE;
    GVL_INTENT_SAFETY.I_Gas_Close_Required := TRUE;
    GVL_INTENT_SAFETY.I_Boiler_Stop_Required := TRUE;
    GVL_INTENT_SAFETY.I_Vent_Force_PV3_Boost := TRUE;
    GVL_INTENT_SAFETY.I_Vent_Force_Supply_100 := TRUE;
END_IF;

IF GVL_HEALTH_BRIDGE.G_CO_Warning_Level OR GVL_HEALTH_BRIDGE.G_CO_Alarm_Level THEN
    GVL_INTENT_SAFETY.I_Vent_Force_Supply_80 := TRUE;
END_IF;

IF GVL_STATE.G_Safety_Leak_Latched THEN
    GVL_INTENT_SAFETY.I_Water_Main_Close_Required := TRUE;
END_IF;

// ========================================
// SAFETY_RESIDUAL_NON_WORKFLOW_PROJECTION
// ========================================
IF GVL_STATE.G_Freeze_Hardware_Degraded THEN
    GVL_INTENT_SAFETY.I_Freeze_Protection_Required := TRUE;
END_IF;

// >>> BULK_SYNC_ANCHOR: PRG_Safety <<<
          
END_PROGRAM

PROGRAM PRG_Test_Scenario_Runner

            IF NOT GVL_TEST.G_Test_Enable THEN
    RETURN;
END_IF;

IF NOT GVL_TEST_INJECTION.G_Scenario_Enable THEN
    RETURN;
END_IF;

// Reset request
IF GVL_TEST_INJECTION.G_Scenario_Reset_Request THEN
    GVL_TEST_INJECTION.G_Inject_Enable := FALSE;
    GVL_TEST_INJECTION.G_Inject_Gas_Level := 0.0;
    GVL_TEST_INJECTION.G_Inject_Force_Gas_Alarm_Reset := FALSE;
    GVL_TEST_INJECTION.G_Inject_Force_IO_Offline := FALSE;
    GVL_TEST_INJECTION.G_Scenario_Step := 0;
    GVL_TEST_INJECTION.G_Scenario_Done := FALSE;
    GVL_TEST_INJECTION.G_Scenario_Failed := FALSE;
    GVL_TEST_INJECTION.G_Scenario_Reset_Request := FALSE;
END_IF;

CASE GVL_TEST_INJECTION.G_Scenario_Current OF

// =========================
// SCENARIO 1: GAS + WATCHDOG
// =========================
1:
    CASE GVL_TEST_INJECTION.G_Scenario_Step OF
    0:
        GVL_TEST_INJECTION.G_Inject_Enable := TRUE;
        GVL_TEST_INJECTION.G_Inject_Gas_Level := 50.0;
        GVL_TEST_INJECTION.G_Scenario_Status_Msg := 'Gas injected';
        GVL_TEST_INJECTION.G_Scenario_Step := 1;

    1:
        GVL_TEST_INJECTION.G_Inject_Force_Gas_Alarm_Reset := TRUE;
        GVL_TEST_INJECTION.G_Scenario_Status_Msg := 'Forced alarm reset';
        GVL_TEST_INJECTION.G_Scenario_Step := 2;

    2:
        IF GVL_TEST.G_Ownership_Violation THEN
            GVL_TEST_INJECTION.G_Scenario_Done := TRUE;
            GVL_TEST_INJECTION.G_Scenario_Status_Msg := 'Watchdog OK';
        ELSE
            GVL_TEST_INJECTION.G_Scenario_Failed := TRUE;
        END_IF;
    END_CASE;

// =========================
// SCENARIO 2: IO OFFLINE
// =========================
2:
    CASE GVL_TEST_INJECTION.G_Scenario_Step OF
    0:
        GVL_TEST_INJECTION.G_Inject_Enable := TRUE;
        GVL_TEST_INJECTION.G_Inject_Force_IO_Offline := TRUE;
        GVL_TEST_INJECTION.G_Scenario_Status_Msg := 'IO offline injected';
        GVL_TEST_INJECTION.G_Scenario_Step := 1;

    1:
        IF NOT GVL_STATUS.G_IO_Modules_Online[1] THEN
            GVL_TEST_INJECTION.G_Scenario_Done := TRUE;
            GVL_TEST_INJECTION.G_Scenario_Status_Msg := 'IO fail-safe OK';
        ELSE
            GVL_TEST_INJECTION.G_Scenario_Failed := TRUE;
        END_IF;
    END_CASE;

END_CASE;

// Auto advance
IF GVL_TEST_INJECTION.G_Scenario_Done AND GVL_TEST_INJECTION.G_Scenario_Auto_Run THEN
    GVL_TEST_INJECTION.G_Scenario_Current := GVL_TEST_INJECTION.G_Scenario_Current + 1;
    GVL_TEST_INJECTION.G_Scenario_Reset_Request := TRUE;
END_IF;
          
END_PROGRAM

PROGRAM PRG_Mode_Manager
  VAR
    fbMode : FB_Mode_Manager;
    L_Last_Mode : E_Behavior_Mode := BEHAVIOR_HOME;
  END_VAR

            fbMode(
    VI_Is_Night := GVL_STATUS.G_Is_Night,
    VI_Away_Request := GVL_MODE.G_Away_Request OR GVL_PRESENCE.G_Auto_Away_Request,
    VI_Maintenance_Request := GVL_MODE.G_Maintenance_Request,
    VI_System_Time_MS := GVL_STATUS.G_System_Time_MS
);

GVL_MODE.G_Current_Behavior_Mode := fbMode.VO_Mode;
GVL_MODE.G_Mode_Code := fbMode.VO_Mode_Code;

IF L_Last_Mode <> fbMode.VO_Mode THEN
    GVL_MODE.G_Mode_Last_Change_TS := GVL_STATUS.G_System_Time_MS;
    L_Last_Mode := fbMode.VO_Mode;
END_IF;
          
END_PROGRAM

PROGRAM PRG_IO_Write
  VAR
    L_i : INT;
  END_VAR

            // 2. ЗАПИСЬ ВЫХОДОВ (GVL_STATE -> GVL_IO)

// 2.1. Отопление (Термоэлектрические приводы)
FOR L_i := 1 TO 8 DO
    GVL_IO.DO_Zone_Valves[L_i] := GVL_STATE.G_Zone_Valves[L_i];
END_FOR;

// 2.2. Коллекторы (Насосы и смесительные клапаны)
FOR L_i := 1 TO GVL_CONSTANTS.C_MAX_MANIFOLDS DO
    GVL_IO.DO_Manifold_Pumps[L_i] := GVL_STATE.G_Manifold_Pumps[L_i];
    GVL_IO.AO_Manifold_Valves[L_i] := REAL_TO_UINT(GVL_STATE.G_Manifold_Valves[L_i] * 1000.0);
END_FOR;

// 2.4. Вентиляция
FOR L_i := 1 TO GVL_CONSTANTS.C_MAX_SUPPLY_FANS DO
    GVL_IO.AO_Supply_Fans[L_i] := REAL_TO_UINT(GVL_STATE.G_Supply_Fans[L_i] * 100.0);
END_FOR;
FOR L_i := 1 TO GVL_CONSTANTS.C_MAX_EXHAUST_FANS DO
    GVL_IO.AO_Exhaust_Fans[L_i] := REAL_TO_UINT(GVL_STATE.G_Exhaust_Fans[L_i] * 100.0);
END_FOR;

// 2.5. ГВС
GVL_IO.DO_DHW_Heating_Pump := GVL_STATE.G_DHW_Heating_Pump;
GVL_IO.DO_DHW_Circ_Pump := GVL_STATE.G_DHW_Circ_Pump;
IF GVL_STATUS.G_Is_Active_PLC THEN
    GVL_IO.DO_Backup_Circulation_Pump := GVL_STATE.G_Backup_Circulation_Pump;
    GVL_IO.DO_Electric_Heater_Enable := GVL_STATE.G_Electric_Heater_Enable;
ELSE
    GVL_IO.DO_Backup_Circulation_Pump := FALSE;
    GVL_IO.DO_Electric_Heater_Enable := FALSE;
END_IF;

// 2.6. Освещение и шторы
FOR L_i := 1 TO 8 DO
    GVL_IO.AO_Lighting_Levels[L_i] := BYTE_TO_UINT(GVL_STATE.G_Lighting_Levels[L_i]) * 10;
END_FOR;
FOR L_i := 1 TO GVL_CONSTANTS.C_MAX_BLINDS DO
    GVL_IO.AO_Blinds_Positions[L_i] := BYTE_TO_UINT(GVL_STATE.G_Blinds_Positions[L_i]) * 10;
END_FOR;

// 2.7. Аварийные выходы (Сирены и клапаны)
GVL_IO.DO_Gas_Siren := (GVL_ALARM.G_Gas_Fire_Siren AND GVL_ALARM.G_Gas_Alarm_Active);
GVL_IO.DO_Fire_Siren := (GVL_ALARM.G_Gas_Fire_Siren AND GVL_ALARM.G_Fire_Alarm_Active);
GVL_IO.DO_Security_Siren := GVL_ALARM.G_Security_Siren;

// === STAGE H2: USE SHADOW COMMANDS ===
GVL_IO.DO_Water_Valve_35_Close := GVL_COMMAND_SHADOW.G_Close_Valve_35;
GVL_IO.DO_Water_Valve_36_Close := GVL_COMMAND_SHADOW.G_Close_Valve_36;
GVL_IO.DO_Gas_Valve_Close := GVL_COMMAND_SHADOW.G_Gas_Valve_Close;

// Access control (shadow)
GVL_IO.DO_Lock_1_Open := GVL_COMMAND_SHADOW.G_Lock_1_Open;
GVL_IO.DO_Lock_1_Close := GVL_COMMAND_SHADOW.G_Lock_1_Close;
GVL_IO.DO_Lock_2_Open := GVL_COMMAND_SHADOW.G_Lock_2_Open;
GVL_IO.DO_Lock_2_Close := GVL_COMMAND_SHADOW.G_Lock_2_Close;

// Gate/Wicket — now via shadow
GVL_IO.DO_Gate_Open := GVL_COMMAND_SHADOW.G_Gate_Open;
GVL_IO.DO_Wicket_Open := GVL_COMMAND_SHADOW.G_Wicket_Open;

// 2.9. Розетки
GVL_IO.DO_Sockets := GVL_STATE.G_Socket_States;

// Selective zonal water recovery outputs
FOR L_i := 1 TO 32 DO
    GVL_IO.DO_Water_Zone_Enable[L_i] := GVL_STATE.G_Water_Zone_Enable[L_i];
END_FOR;

// >>> BULK_SYNC_ANCHOR: PRG_IO_Write <<<
          
END_PROGRAM

PROGRAM PRG_Command_Verifier
  VAR
    L_Mismatch_Count : INT := 0;
  END_VAR

            // Current-cycle mismatch count between legacy and shadow command layers
L_Mismatch_Count := 0;

IF GVL_COMMAND.G_Gas_Valve_Close <> GVL_COMMAND_SHADOW.G_Gas_Valve_Close THEN
    L_Mismatch_Count := L_Mismatch_Count + 1;
END_IF;

IF GVL_COMMAND.G_Boiler_Stop <> GVL_COMMAND_SHADOW.G_Boiler_Stop THEN
    L_Mismatch_Count := L_Mismatch_Count + 1;
END_IF;

IF GVL_COMMAND.G_Vent_Stop <> GVL_COMMAND_SHADOW.G_Vent_Stop THEN
    L_Mismatch_Count := L_Mismatch_Count + 1;
END_IF;

IF GVL_COMMAND.G_Supply_100_Req <> GVL_COMMAND_SHADOW.G_Supply_100_Req THEN
    L_Mismatch_Count := L_Mismatch_Count + 1;
END_IF;

IF GVL_COMMAND.G_Supply_80_Req <> GVL_COMMAND_SHADOW.G_Supply_80_Req THEN
    L_Mismatch_Count := L_Mismatch_Count + 1;
END_IF;

IF GVL_COMMAND.G_Vent_PV3_Boost <> GVL_COMMAND_SHADOW.G_Vent_PV3_Boost THEN
    L_Mismatch_Count := L_Mismatch_Count + 1;
END_IF;

IF GVL_COMMAND.G_Close_Valve_35 <> GVL_COMMAND_SHADOW.G_Close_Valve_35 THEN
    L_Mismatch_Count := L_Mismatch_Count + 1;
END_IF;

IF GVL_COMMAND.G_Close_Valve_36 <> GVL_COMMAND_SHADOW.G_Close_Valve_36 THEN
    L_Mismatch_Count := L_Mismatch_Count + 1;
END_IF;

IF GVL_COMMAND.G_Lock_1_Open <> GVL_COMMAND_SHADOW.G_Lock_1_Open THEN
    L_Mismatch_Count := L_Mismatch_Count + 1;
END_IF;

IF GVL_COMMAND.G_Lock_1_Close <> GVL_COMMAND_SHADOW.G_Lock_1_Close THEN
    L_Mismatch_Count := L_Mismatch_Count + 1;
END_IF;

IF GVL_COMMAND.G_Lock_2_Open <> GVL_COMMAND_SHADOW.G_Lock_2_Open THEN
    L_Mismatch_Count := L_Mismatch_Count + 1;
END_IF;

IF GVL_COMMAND.G_Lock_2_Close <> GVL_COMMAND_SHADOW.G_Lock_2_Close THEN
    L_Mismatch_Count := L_Mismatch_Count + 1;
END_IF;

// Gate and wicket comparison
IF GVL_COMMAND.G_Gate_Open <> GVL_COMMAND_SHADOW.G_Gate_Open THEN
    L_Mismatch_Count := L_Mismatch_Count + 1;
END_IF;

IF GVL_COMMAND.G_Wicket_Open <> GVL_COMMAND_SHADOW.G_Wicket_Open THEN
    L_Mismatch_Count := L_Mismatch_Count + 1;
END_IF;

GVL_COMMAND_VERIFY.Command_Mismatch_Count := L_Mismatch_Count;
GVL_COMMAND_VERIFY.Command_Match_OK := (L_Mismatch_Count = 0);
GVL_COMMAND_VERIFY.Command_Mismatch_Active := (L_Mismatch_Count > 0);
          
END_PROGRAM

PROGRAM PRG_Presence_Manager
  VAR
    fbPresence : FB_Presence_Manager;
    L_i : INT;
  END_VAR

            fbPresence(
    VI_Motion_Sensors := GVL_STATE.G_Motion_Sensors,
    VI_System_Time_MS := GVL_STATUS.G_System_Time_MS
);

GVL_PRESENCE.G_Any_Motion := fbPresence.VO_Any_Motion;
GVL_PRESENCE.G_Occupied := fbPresence.VO_Occupied;
GVL_PRESENCE.G_Auto_Away_Request := fbPresence.VO_Auto_Away;
GVL_PRESENCE.G_Last_Motion_TS := fbPresence.VO_Last_Motion_TS;

FOR L_i := 1 TO GVL_CONSTANTS.C_MAX_ZONES DO
    IF GVL_STATE.G_Motion_Sensors[L_i] THEN
        GVL_PRESENCE.G_Zone_Occupied[L_i] := TRUE;
        GVL_PRESENCE.G_Zone_Last_Motion_TS[L_i] := GVL_STATUS.G_System_Time_MS;
    END_IF;

    IF (GVL_STATUS.G_System_Time_MS - GVL_PRESENCE.G_Zone_Last_Motion_TS[L_i]) > 900000 THEN
        GVL_PRESENCE.G_Zone_Occupied[L_i] := FALSE;
    END_IF;
END_FOR;
          
END_PROGRAM

PROGRAM PRG_Test_Injection

            // Non-intrusive test injection layer
// Must be called AFTER PRG_IO_Read and BEFORE PRG_Safety

IF NOT GVL_TEST_INJECTION.G_Inject_Enable THEN
    RETURN;
END_IF;

// ===== GAS INJECTION =====
IF GVL_TEST_INJECTION.G_Inject_Gas_Level > 0.0 THEN
    GVL_STATE.G_Methane_Sensors[1] := GVL_TEST_INJECTION.G_Inject_Gas_Level;
END_IF;

// ===== IO OFFLINE INJECTION =====
IF GVL_TEST_INJECTION.G_Inject_Force_IO_Offline THEN
    GVL_STATUS.G_IO_Modules_Online[1] := FALSE;
    GVL_STATUS.G_IO_Modules_Online[2] := FALSE;
END_IF;

// ===== OWNERSHIP VIOLATION TEST =====
// Intentionally break safety to verify watchdog
IF GVL_TEST_INJECTION.G_Inject_Force_Gas_Alarm_Reset THEN
    GVL_STATE.G_Safety_Gas_Alarm := FALSE;
END_IF;
          
END_PROGRAM

PROGRAM PRG_Lighting
  VAR
    L_i : INT;
    fbLightingManager : FB_Lighting_Blinds_Manager;
    fbSocketManager : FB_Socket_Manager;
    L_Manual_Light_Override_32 : ARRAY[1..32] OF BYTE;
    L_Manual_Blinds_Override_32 : ARRAY[1..32] OF BYTE;
    L_Manual_Socket_Override_32 : ARRAY[1..32] OF BOOL;
    L_Sim_Lights_32 : ARRAY[1..32] OF BOOL;
    L_Physical_Switches_32 : ARRAY[1..32] OF BOOL;
    L_Motion_Sensors_32 : ARRAY[1..32] OF BOOL;
    L_Blinds_Override : ARRAY[1..GVL_CONSTANTS.C_MAX_BLINDS] OF BYTE;
    L_Socket_Override : ARRAY[1..GVL_CONSTANTS.C_MAX_SOCKETS] OF BOOL;
  END_VAR

            FOR L_i := 1 TO 32 DO
    IF L_i <= 16 THEN
        IF GVL_INTENT_SYSTEM.I_Lighting_Overrides_Block OR GVL_SYSTEM_COORDINATION.G_Block_Lighting_Override THEN
            L_Manual_Light_Override_32[L_i] := 0;
        ELSE
            L_Manual_Light_Override_32[L_i] := GVL_INTENT_USER.I_Lighting_Override_32[L_i];
        END_IF;
        L_Sim_Lights_32[L_i] := GVL_STATE.G_Sim_Lights[L_i];
        L_Physical_Switches_32[L_i] := GVL_STATE.G_Physical_Switches[L_i];
        L_Motion_Sensors_32[L_i] := GVL_STATE.G_Motion_Sensors[L_i];
    ELSE
        L_Manual_Light_Override_32[L_i] := 0;
        L_Sim_Lights_32[L_i] := FALSE;
        L_Physical_Switches_32[L_i] := FALSE;
        L_Motion_Sensors_32[L_i] := FALSE;
    END_IF;

    IF GVL_INTENT_SYSTEM.I_Blinds_Overrides_Block THEN
        L_Manual_Blinds_Override_32[L_i] := 0;
    ELSE
        L_Manual_Blinds_Override_32[L_i] := GVL_INTENT_USER.I_Blinds_Override_32[L_i];
    END_IF;

    IF GVL_INTENT_SYSTEM.I_Socket_Overrides_Block OR GVL_SYSTEM_COORDINATION.G_Block_Sockets_Override THEN
        L_Manual_Socket_Override_32[L_i] := FALSE;
    ELSE
        L_Manual_Socket_Override_32[L_i] := GVL_INTENT_USER.I_Socket_Override_32[L_i];
    END_IF;
END_FOR;

// ADAPTER: copy to FB-sized arrays
FOR L_i := 1 TO GVL_CONSTANTS.C_MAX_BLINDS DO
    L_Blinds_Override[L_i] := L_Manual_Blinds_Override_32[L_i];
END_FOR;

FOR L_i := 1 TO GVL_CONSTANTS.C_MAX_SOCKETS DO
    L_Socket_Override[L_i] := L_Manual_Socket_Override_32[L_i];
END_FOR;

// 10. Управление освещением и шторами
fbLightingManager(
    VI_System_Time_MS := GVL_STATUS.G_System_Time_MS,
    VI_IsActivePLC := GVL_STATUS.G_Is_Active_PLC,
    VI_Current_Scenario := GVL_STATUS.G_Current_Scenario,
    VI_Away_Level := 1,
    VI_Simulation_Active := GVL_STATUS.G_Sim_Active,
    VI_Manual_Light_Override := L_Manual_Light_Override_32,
    VI_Manual_Blinds_Override := L_Blinds_Override,
    VI_Simulation_Lights := L_Sim_Lights_32,
    VI_Physical_Switches := L_Physical_Switches_32,
    VI_Motion_Sensors := L_Motion_Sensors_32,
    VI_Is_Night := GVL_STATUS.G_Is_Night,
    VI_Rule_Actions := GVL_STATE.G_Rule_Actions,
    VI_IO_Modules_Online := GVL_STATUS.G_IO_Modules_Online,
    VI_Wet_Zone_Map := GVL_CONFIG.G_Wet_Zone_Map,
    VI_Scenario_Configs := GVL_CONFIG.G_HMI_Scenario_Configs,
    VO_Lighting_Levels => GVL_STATE.G_Lighting_Levels,
    VO_Blinds_Positions => GVL_STATE.G_Blinds_Positions
);

// 11.5 Управление розетками
fbSocketManager(
    VI_System_Time_MS := GVL_STATUS.G_System_Time_MS,
    VI_IsActivePLC := GVL_STATUS.G_Is_Active_PLC,
    VI_Scenario := GVL_STATUS.G_Current_Scenario,
    VI_Manual_Override := L_Socket_Override,
    VI_Physical_Switches := GVL_STATE.G_Socket_Switches,
    VI_Rule_Actions := GVL_STATE.G_Rule_Actions,
    VI_Fire_Alarm := GVL_ALARM.G_Fire_Alarm_Active,
    VI_Flood_Alarm := GVL_ALARM.G_Flood_Alarm_Active,
    VI_Security_Armed := GVL_ALARM.G_Security_Armed,
    VI_IO_Modules_Online := GVL_STATUS.G_IO_Modules_Online,
    VO_Socket_States => GVL_STATE.G_Socket_States
);

// Evacuation lighting override
IF GVL_STATE.G_Evacuation_Lighting_Active THEN
    FOR L_i := 1 TO 8 DO
        IF (L_i MOD 2) = 0 THEN
            GVL_STATE.G_Lighting_Levels[L_i] := 100;
        ELSE
            GVL_STATE.G_Lighting_Levels[L_i] := 0;
        END_IF;
    END_FOR;
END_IF;

// Directional evacuation override
IF GVL_STATE.G_Evacuation_Lighting_Active THEN
    FOR L_i := 1 TO GVL_CONFIG.C_MAX_LIGHT_ZONES DO
        CASE GVL_STATE.G_Evac_Guidance[L_i] OF
            -1:
                GVL_STATE.G_Lighting_Levels[L_i] := 0;
            1:
                GVL_STATE.G_Lighting_Levels[L_i] := 100;
        ELSE
            GVL_STATE.G_Lighting_Levels[L_i] := SEL((L_i MOD 2) = 0, 0, 100);
        END_CASE;
    END_FOR;
END_IF;
// >>> BULK_SYNC_ANCHOR: PRG_Lighting <<<
          
END_PROGRAM

PROGRAM PRG_Security
  VAR
    L_i : INT;
    L_Motion_Sensors_16 : ARRAY[1..16] OF BOOL;
    fbSecurityManager : FB_Security_System_Manager;
    fbAccessControl : FB_Access_Control;
  END_VAR

            FOR L_i := 1 TO 16 DO
    L_Motion_Sensors_16[L_i] := GVL_STATE.G_Motion_Sensors[L_i];
END_FOR;
// 7. Система безопасности (Охранная сигнализация)
fbSecurityManager(
    VI_System_Time_MS := GVL_STATUS.G_System_Time_MS,
    VI_IsActivePLC := GVL_STATUS.G_Is_Active_PLC,
    VI_Motion_Sensors := L_Motion_Sensors_16,
    VI_Door_Sensors := GVL_STATE.G_Door_Sensors,
    VI_Window_Sensors := GVL_STATE.G_Window_Sensors,
    VI_Arm_Request := GVL_INTENT_USER.I_Arm_Request,
    VI_Disarm_Request := GVL_INTENT_USER.I_Disarm_Request,
    VI_PIN_Code := GVL_INTENT_USER.I_PIN_Code,
    VI_RFID_Tag := GVL_INTENT_USER.I_RFID_Tag,
    VI_2FA_Code := GVL_INTENT_USER.I_2FA_Code_In,
    VI_Config := GVL_CONFIG.G_Security_Config,
    VI_Bypass_Motion := GVL_CONFIG.G_Security_Config.bypass_motion,
    VI_Bypass_Doors := GVL_CONFIG.G_Security_Config.bypass_doors,
    VI_Bypass_Windows := GVL_CONFIG.G_Security_Config.bypass_windows,
    VI_Current_TOD := GVL_STATUS.G_Current_TOD,
    VO_Armed => GVL_ALARM.G_Security_Armed,
    VO_Alarm_Active => GVL_ALARM.G_Security_Alarm,
    VO_Siren_Active => GVL_ALARM.G_Security_Siren,
    VO_Status_Msg => GVL_STATUS.G_Security_Status_Msg,
    VO_Send_Code_Req => GVL_COMMAND.G_Send_2FA_Req,
    VO_Code_To_Send => GVL_COMMAND.G_2FA_Code_Out
);

// 7.1 Контроль доступа (СКУД)
fbAccessControl(
    VI_System_Time_MS := GVL_STATUS.G_System_Time_MS,
    VI_IsActivePLC := GVL_STATUS.G_Is_Active_PLC,
    VI_Armed := GVL_ALARM.G_Security_Armed,
    VI_System_Mode := GVL_STATE.G_System_Mode,
    VI_Gate_Open_Req := GVL_CONFIG.G_HMI_Gate_Open_Req,
    VI_Wicket_Open_Req := GVL_CONFIG.G_HMI_Wicket_Open_Req,
    VI_Lock_1_Open_Req := GVL_CONFIG.G_HMI_Lock_1_Open_Req,
    VI_Lock_1_Close_Req := GVL_CONFIG.G_HMI_Lock_1_Close_Req,
    VI_Lock_2_Open_Req := GVL_CONFIG.G_HMI_Lock_2_Open_Req,
    VI_Lock_2_Close_Req := GVL_CONFIG.G_HMI_Lock_2_Close_Req,
    VI_PIN_Code := GVL_INTENT_USER.I_PIN_Code,
    VI_RFID_Tag := GVL_INTENT_USER.I_RFID_Tag,
    VI_Access_Codes := GVL_Retain.G_Access_Codes,
    VI_RFID_Tags := GVL_Retain.G_RFID_Tags,
    VI_Config := GVL_CONFIG.G_Security_Config,
    VO_Gate_Open => GVL_INTENT_USER.I_Gate_Open_Request,
    VO_Wicket_Open => GVL_INTENT_USER.I_Wicket_Open_Request,
    VO_Lock_1_Open => GVL_INTENT_USER.I_Lock_1_Open_Request,
    VO_Lock_1_Close => GVL_INTENT_USER.I_Lock_1_Close_Request,
    VO_Lock_2_Open => GVL_INTENT_USER.I_Lock_2_Open_Request,
    VO_Lock_2_Close => GVL_INTENT_USER.I_Lock_2_Close_Request
);
          
END_PROGRAM

PROGRAM PRG_System_Coordinator
  VAR
    fbCoord : FB_System_Coordinator;
  END_VAR

            fbCoord(
    VI_Fire_Latched := GVL_STATE.G_Safety_Smoke_Latched,
    VI_Gas_Latched := GVL_STATE.G_Safety_Gas_Latched,
    VI_Leak_Latched := GVL_STATE.G_Safety_Leak_Latched,
    VI_IO_Degraded := NOT GVL_STATUS.G_IO_Modules_Online[1],
    VI_Ownership_Violation := GVL_TEST.G_Ownership_Violation,
    VI_Behavior_Mode := GVL_MODE.G_Current_Behavior_Mode
);

GVL_SYSTEM_COORDINATION.G_Block_Heating := fbCoord.VO_Block_Heating;
GVL_SYSTEM_COORDINATION.G_Block_Ventilation := fbCoord.VO_Block_Ventilation;
GVL_SYSTEM_COORDINATION.G_Block_Lighting_Override := fbCoord.VO_Block_Lighting;
GVL_SYSTEM_COORDINATION.G_Block_Sockets_Override := fbCoord.VO_Block_Sockets;

GVL_SYSTEM_COORDINATION.G_System_Degraded := fbCoord.VO_System_Degraded;
GVL_SYSTEM_COORDINATION.G_Coordination_Code := fbCoord.VO_Code;
          
END_PROGRAM

PROGRAM PRG_Heating
  VAR
    L_Last_Mode : INT := 0;
    L_Mode_Hold_Timer : FB_System_Timer;
  END_VAR
  VAR
    fbHeatingManager : FB_Heating_System_Manager;
    fbDHWManager : FB_DHW_Manager;
    fbDiagEventManager : FB_Diagnostics_Event_Manager;
    fbDecision : FB_Heating_Decision_Context;
    L_i : INT;
    L_j : INT;
    L_Zone_ID : INT;
    L_Zone_Valves : ARRAY[1..GVL_CONSTANTS.C_MAX_HEATING_CIRCUITS] OF BOOL;
    L_Boiler_Modulation_REAL : ARRAY[1..GVL_CONSTANTS.C_MAX_BOILERS] OF REAL;
    L_Heating_Emergency_Stop : BOOL;
    L_Heating_Gas_Safety_Stop : BOOL;
    L_Heating_DHW_Demand : BOOL;
    L_Manifold_Adjusted_Priority : ARRAY[1..GVL_CONSTANTS.C_MAX_MANIFOLDS] OF INT;
  END_VAR

            // ============================================================
// S1. INPUTS / LOCAL ARBITRATION CONTEXT
// ============================================================

FOR L_i := 1 TO GVL_CONSTANTS.C_MAX_BOILERS DO
    L_Boiler_Modulation_REAL[L_i] := TO_REAL(GVL_IO.AI_Boiler_Modulation[L_i]);
END_FOR;

L_Heating_Emergency_Stop := GVL_STATE.G_Safety_Emergency_Stop;
L_Heating_Gas_Safety_Stop := GVL_STATE.G_Safety_Gas_Latched;
L_Heating_DHW_Demand := fbDHWManager.VO_Heating_Pump;

IF L_Heating_Emergency_Stop THEN
    L_Heating_Gas_Safety_Stop := FALSE;
    L_Heating_DHW_Demand := FALSE;
ELSIF L_Heating_Gas_Safety_Stop THEN
    L_Heating_DHW_Demand := FALSE;
ELSIF GVL_STATE.G_System_Mode = E_System_Operating_Mode.MODE_DEGRADED THEN
    L_Heating_DHW_Demand := FALSE;
END_IF;

L_Mode_Hold_Timer(
    IN := TRUE,
    PT := T#30s,
    VI_System_Time_MS := GVL_STATUS.G_System_Time_MS
);

IF L_Mode_Hold_Timer.Q THEN
    IF GVL_STATE.G_Freeze_Request THEN
        L_Last_Mode := 2;
    ELSIF GVL_STATE.G_Preheat_Request THEN
        L_Last_Mode := 1;
    ELSE
        L_Last_Mode := 0;
    END_IF;
END_IF;

CASE L_Last_Mode OF
    2: GVL_STATE.G_Target_Temperature := 5.0;
    1: GVL_STATE.G_Target_Temperature := 22.0;
    ELSE GVL_STATE.G_Target_Temperature := 20.0;
END_CASE;

// ============================================================
// S1.5 DECISION CONTEXT / THERMAL ALLOCATION
// ============================================================

// === HP-1 + HP-2 PRIORITY BIAS APPLICATION ===
FOR L_i := 1 TO GVL_CONSTANTS.C_MAX_MANIFOLDS DO
    L_Manifold_Adjusted_Priority[L_i] := GVL_CONFIG.G_Manifold_Priority[L_i];
END_FOR;

FOR L_i := 1 TO GVL_CONSTANTS.C_MAX_HEATING_CIRCUITS DO
    L_j := TO_INT(GVL_CONFIG.G_HMI_FloorHeating_Configs[L_i].manifold_id);
    L_Zone_ID := GVL_CONFIG.G_Heating_Circuit_To_Zone[L_i];

    IF (L_j >= 1) AND (L_j <= GVL_CONSTANTS.C_MAX_MANIFOLDS) AND (L_Zone_ID >= 1) AND (L_Zone_ID <= GVL_CONSTANTS.C_MAX_ZONES) THEN

        // Base policy bias (HP-1), mapped circuit -> logical zone
        L_Manifold_Adjusted_Priority[L_j] := L_Manifold_Adjusted_Priority[L_j] + TO_INT(GVL_HEATING_POLICY.G_Zone_Priority_Bias[L_Zone_ID]);

        // Guest preheat boost (HP-2, config-driven), mapped circuit -> logical zone
        IF GVL_HEATING_POLICY_CONFIG.G_Guest_Preheat_Enabled AND GVL_HEATING_POLICY.G_Zone_Guest_Preheat_Request[L_Zone_ID] THEN
            L_Manifold_Adjusted_Priority[L_j] := L_Manifold_Adjusted_Priority[L_j] + GVL_HEATING_POLICY_CONFIG.G_Guest_Preheat_Priority_Boost;
        END_IF;

        // Lower bound
        IF L_Manifold_Adjusted_Priority[L_j] < 1 THEN
            L_Manifold_Adjusted_Priority[L_j] := 1;
        END_IF;

    END_IF;
END_FOR;

fbDecision(
    VI_Manifold_Pump_In_Service := GVL_CONFIG.G_Manifold_Pump_In_Service,
    VI_Manifold_Pressure_Fault := GVL_STATUS.G_Diagnostics.Manifold_Pressure_Fault,
    VI_Manifold_Current_Fault := GVL_STATUS.G_Diagnostics.Manifold_Current_Fault,
    VI_Manifold_Thermal_Weight := GVL_CONFIG.G_Manifold_Thermal_Weight,
    VI_Manifold_Priority := L_Manifold_Adjusted_Priority,
    VI_Max_Thermal_Budget := GVL_CONFIG.G_Max_Thermal_Budget
);

// ============================================================
// S2. HEATING / DHW ORCHESTRATION CALLS
// ============================================================

fbHeatingManager(
    VI_Preheat_Request := GVL_STATE.G_Preheat_Request,
    VI_System_Time_MS := GVL_STATUS.G_System_Time_MS,
    VI_Current_TOD := GVL_STATUS.G_Current_TOD,
    VI_IsActivePLC := GVL_STATUS.G_Is_Active_PLC,
    VI_Outdoor_Temp := GVL_STATE.G_Outdoor_Temp,
    VI_Floor_Temps := GVL_STATE.G_Floor_Temps,
    VI_Room_Temps := GVL_STATE.G_Room_Temps,
    VI_Config := GVL_CONFIG.G_Heating_Config,
    VI_Zone_Configs := GVL_CONFIG.G_HMI_FloorHeating_Configs,
    VI_Tariff := GVL_CONFIG.G_HMI_Tariff_Settings,
    VI_Current_Hour := TO_UINT(GVL_STATUS.G_Time_Of_Day_MS / GVL_CONSTANTS.C_MS_IN_HOUR),
    VI_Manifold_Pressures := GVL_STATE.G_Manifold_Pressures,
    VI_Manifold_Currents := GVL_STATE.G_Manifold_Currents,
    VI_Manifold_Temps_Supply := GVL_STATE.G_Manifold_T_Supply,
    VI_Manifold_Temps_Return := GVL_STATE.G_Manifold_T_Return,
    VI_Boiler_Flame_Status := GVL_STATE.G_Boiler_Flame,
    VI_Boiler_Error_Status := GVL_STATE.G_Boiler_Error,
    VI_Boiler_OT_Online := GVL_STATE.G_Boiler_OT_Online,
    VI_Boiler_Modulation := L_Boiler_Modulation_REAL,
    VI_Rule_Actions := GVL_STATE.G_Rule_Actions,
    VI_Boiler_Stop := FALSE,
    VI_IO_Modules_Online := GVL_STATUS.G_IO_Modules_Online,
    VI_DHW_Heating_Demand := L_Heating_DHW_Demand,
    VI_DHW_Target_Temp := GVL_CONFIG.G_DHW_Config.Target_Temp,
    VI_Current_Scenario := GVL_STATUS.G_Current_Scenario,
    VI_System_Mode := GVL_STATE.G_System_Mode,
    VI_Emergency_Stop := L_Heating_Emergency_Stop,
    VI_Gas_Safety_Stop := L_Heating_Gas_Safety_Stop,
    VI_Scenario_Configs := GVL_CONFIG.G_HMI_Scenario_Configs,
    VI_Manifold_End_Switches := GVL_STATE.G_Manifold_End_Switches,
    VI_Valve_Test_Config := GVL_CONFIG.G_Valve_Test_Config,
    VO_Manifold_Valves => GVL_STATE.G_Manifold_Valves,
    VO_Manifold_Pumps => GVL_STATE.G_Manifold_Pumps,
    VO_Zone_Valves => L_Zone_Valves,
    VO_Boiler_OT_Enable => GVL_STATE.G_Boiler_OT_Enable,
    VO_Boiler_OT_Setpoint => GVL_STATE.G_Boiler_OT_Setpoint,
    VO_Backup_Circulation_Pump => GVL_STATE.G_Backup_Circulation_Pump,
    VO_Electric_Heater_Enable => GVL_STATE.G_Electric_Heater_Enable,
    VO_Freeze_Risk_Status => GVL_STATE.G_Safety_Freeze_Risk,
    VO_Status => GVL_STATUS.G_Manifold_Status,
    VO_Boiler_Status => GVL_STATUS.G_Boiler_Status
);

// Apply global and thermal allocation constraints after base heating orchestration.
// Coordinator owns cross-subsystem blocking; decision context owns eligibility/budget.
// Heating manager remains the control algorithm owner.
FOR L_i := 1 TO GVL_CONSTANTS.C_MAX_MANIFOLDS DO
    IF GVL_SYSTEM_COORDINATION.G_Block_Heating OR (NOT fbDecision.VO_Manifold_Enabled[L_i]) THEN
        GVL_STATE.G_Manifold_Pumps[L_i] := FALSE;
        GVL_STATE.G_Manifold_Valves[L_i] := 0.0;

        FOR L_j := 1 TO GVL_CONSTANTS.C_MAX_HEATING_CIRCUITS DO
            IF GVL_CONFIG.G_HMI_FloorHeating_Configs[L_j].manifold_id = L_i THEN
                L_Zone_Valves[L_j] := FALSE;
            END_IF;
        END_FOR;
    END_IF;
END_FOR;

fbDHWManager(
    VI_System_Time_MS := GVL_STATUS.G_System_Time_MS,
    VI_Current_TOD := GVL_STATUS.G_Current_TOD,
    VI_IsActivePLC := GVL_STATUS.G_Is_Active_PLC,
    VI_Temp := GVL_STATE.G_DHW_Temp,
    VI_Pressure := GVL_STATE.G_DHW_Pressure,
    VI_Config := GVL_CONFIG.G_DHW_Config,
    VI_Current_Day_Of_Week := GVL_STATUS.G_Current_Day,
    VI_IO_Modules_Online := GVL_STATUS.G_IO_Modules_Online,
    VI_Reset_Errors := GVL_INTENT_USER.I_Reset_Errors,
    VI_Emergency_Stop := GVL_STATE.G_Safety_Emergency_Stop,
    VI_System_Mode := GVL_STATE.G_System_Mode,
    VO_Heating_Pump => GVL_STATE.G_DHW_Heating_Pump,
    VO_Circ_Pump => GVL_STATE.G_DHW_Circ_Pump,
    VO_Status => GVL_STATUS.G_DHW_Status
);

// ============================================================
// S3. DIAGNOSTICS PROJECTION + EVENTS
// ============================================================

GVL_STATUS.G_Diagnostics.Backup_Pump_Out_Of_Service := NOT GVL_CONFIG.G_Backup_Circulation_Pump_In_Service;
GVL_STATUS.G_Diagnostics.Electric_Heater_Out_Of_Service := NOT GVL_CONFIG.G_Electric_Heater_In_Service;

fbDiagEventManager(
    VI_Code := GVL_CONFIG.ERR_BACKUP_PUMP_OUT_OF_SERVICE,
    VI_Severity := 2,
    VI_Active := NOT GVL_CONFIG.G_Backup_Circulation_Pump_In_Service,
    VI_Timestamp := GVL_STATUS.G_System_Time_MS,
    VI_Source := 400,
    VIO_Events := GVL_STATUS.G_Diagnostics_Events,
    VIO_Count := GVL_STATUS.G_Diagnostics_Count
);

fbDiagEventManager(
    VI_Code := GVL_CONFIG.ERR_ELECTRIC_HEATER_OUT_OF_SERVICE,
    VI_Severity := 2,
    VI_Active := NOT GVL_CONFIG.G_Electric_Heater_In_Service,
    VI_Timestamp := GVL_STATUS.G_System_Time_MS,
    VI_Source := 401,
    VIO_Events := GVL_STATUS.G_Diagnostics_Events,
    VIO_Count := GVL_STATUS.G_Diagnostics_Count
);

FOR L_i := 1 TO GVL_CONSTANTS.C_MAX_MANIFOLDS DO
    GVL_STATUS.G_Diagnostics.Manifold_Pump_Out_Of_Service[L_i] := NOT GVL_CONFIG.G_Manifold_Pump_In_Service[L_i];

    fbDiagEventManager(
        VI_Code := GVL_CONFIG.ERR_MANIFOLD_PUMP_OUT_OF_SERVICE,
        VI_Severity := 2,
        VI_Active := NOT GVL_CONFIG.G_Manifold_Pump_In_Service[L_i],
        VI_Timestamp := GVL_STATUS.G_System_Time_MS,
        VI_Source := 410 + L_i,
        VIO_Events := GVL_STATUS.G_Diagnostics_Events,
        VIO_Count := GVL_STATUS.G_Diagnostics_Count
    );
END_FOR;

GVL_STATUS.G_Diagnostics.DHW_Heating_Pump_Out_Of_Service := NOT GVL_CONFIG.G_DHW_Heating_Pump_In_Service;
GVL_STATUS.G_Diagnostics.DHW_Circ_Pump_Out_Of_Service := NOT GVL_CONFIG.G_DHW_Circ_Pump_In_Service;

fbDiagEventManager(
    VI_Code := GVL_CONFIG.ERR_DHW_HEATING_PUMP_OUT_OF_SERVICE,
    VI_Severity := 2,
    VI_Active := NOT GVL_CONFIG.G_DHW_Heating_Pump_In_Service,
    VI_Timestamp := GVL_STATUS.G_System_Time_MS,
    VI_Source := 420,
    VIO_Events := GVL_STATUS.G_Diagnostics_Events,
    VIO_Count := GVL_STATUS.G_Diagnostics_Count
);

fbDiagEventManager(
    VI_Code := GVL_CONFIG.ERR_DHW_CIRC_PUMP_OUT_OF_SERVICE,
    VI_Severity := 2,
    VI_Active := NOT GVL_CONFIG.G_DHW_Circ_Pump_In_Service,
    VI_Timestamp := GVL_STATUS.G_System_Time_MS,
    VI_Source := 421,
    VIO_Events := GVL_STATUS.G_Diagnostics_Events,
    VIO_Count := GVL_STATUS.G_Diagnostics_Count
);

fbDiagEventManager(
    VI_Code := GVL_CONFIG.ERR_FREEZE_HARDWARE_FAILED,
    VI_Severity := 4,
    VI_Active := GVL_STATE.G_Freeze_Hardware_Failed,
    VI_Timestamp := GVL_STATUS.G_System_Time_MS,
    VI_Source := 430,
    VIO_Events := GVL_STATUS.G_Diagnostics_Events,
    VIO_Count := GVL_STATUS.G_Diagnostics_Count
);

// ============================================================
// S4. MAINTENANCE GATING
// ============================================================

IF NOT GVL_CONFIG.G_Backup_Circulation_Pump_In_Service THEN
    GVL_STATE.G_Backup_Circulation_Pump := FALSE;
END_IF;
IF NOT GVL_CONFIG.G_Electric_Heater_In_Service THEN
    GVL_STATE.G_Electric_Heater_Enable := FALSE;
END_IF;
FOR L_i := 1 TO GVL_CONSTANTS.C_MAX_MANIFOLDS DO
    IF NOT GVL_CONFIG.G_Manifold_Pump_In_Service[L_i] THEN
        GVL_STATE.G_Manifold_Pumps[L_i] := FALSE;
    END_IF;
END_FOR;
IF NOT GVL_CONFIG.G_DHW_Heating_Pump_In_Service THEN
    GVL_STATE.G_DHW_Heating_Pump := FALSE;
END_IF;
IF NOT GVL_CONFIG.G_DHW_Circ_Pump_In_Service THEN
    GVL_STATE.G_DHW_Circ_Pump := FALSE;
END_IF;

// ============================================================
// S5. FREEZE HARDWARE SUPPORT LOGIC
// ============================================================

GVL_STATE.G_Freeze_Hardware_Degraded := GVL_STATUS.G_Diagnostics.Backup_Pump_Fault OR GVL_STATUS.G_Diagnostics.Electric_Heater_Fault;
GVL_STATE.G_Freeze_Hardware_Failed := GVL_STATUS.G_Diagnostics.Backup_Pump_Fault AND GVL_STATUS.G_Diagnostics.Electric_Heater_Fault;
IF GVL_STATE.G_Freeze_Hardware_Failed THEN
    GVL_STATE.G_Backup_Circulation_Pump := FALSE;
    GVL_STATE.G_Electric_Heater_Enable := FALSE;
    GVL_STATE.G_Safety_Freeze_Risk := TRUE;
END_IF;

// >>> BULK_SYNC_ANCHOR: PRG_Heating <<<

// ============================================================
// S6. ADAPTER COPY-OUT
// ============================================================

FOR L_i := 1 TO GVL_CONSTANTS.C_MAX_HEATING_CIRCUITS DO
    GVL_STATE.G_Zone_Valves[L_i] := L_Zone_Valves[L_i];
END_FOR;
          
END_PROGRAM

PROGRAM PRG_IO_Read
  VAR
    L_i : INT;
    L_Debounce_Time : TIME := T#100MS;
    L_Manifold_Pressure_Raw : WORD;
    L_Manifold_Current_Raw : WORD;
    fbDebounce_Switches : ARRAY[1..8] OF FB_System_Timer;
    fbDebounce_Motion : ARRAY[1..8] OF FB_System_Timer;
    fbDebounce_Security_Open : ARRAY[1..GVL_CONSTANTS.C_MAX_SECURITY_SENSORS] OF FB_System_Timer;
    fbDebounce_Security_Glass : ARRAY[1..GVL_CONSTANTS.C_MAX_SECURITY_SENSORS] OF FB_System_Timer;
    fbDebounce_Flood : ARRAY[1..GVL_CONSTANTS.C_MAX_FLOOD_SENSORS] OF FB_System_Timer;
    fbDebounce_Smoke : ARRAY[1..GVL_CONSTANTS.C_MAX_SMOKE_SENSORS] OF FB_System_Timer;
    fbDebounce_Group_2F : FB_System_Timer;
    fbIO_Watchdog_1 : FB_IO_Module_Watchdog;
    fbIO_Watchdog_2 : FB_IO_Module_Watchdog;
    fbDiagEventManager : FB_Diagnostics_Event_Manager;
    L_IO_Error_Active : BOOL;
    fbCalib_Outdoor_Temp : FB_Sensor_Calibration_Processor;
    fbCalib_Supply_Temps : ARRAY[1..GVL_CONSTANTS.C_MAX_SUPPLY_TEMPS] OF FB_Sensor_Calibration_Processor;
    fbCalib_Room_Temps : ARRAY[1..GVL_CONSTANTS.C_MAX_ZONES] OF FB_Sensor_Calibration_Processor;
    fbCalib_Floor_Temps : ARRAY[1..GVL_CONSTANTS.C_MAX_ZONES] OF FB_Sensor_Calibration_Processor;
    fbCalib_Room_Hum : ARRAY[1..GVL_CONSTANTS.C_MAX_ZONES] OF FB_Sensor_Calibration_Processor;
    fbCalib_Room_CO2 : ARRAY[1..GVL_CONSTANTS.C_MAX_ZONES] OF FB_Sensor_Calibration_Processor;
    fbCalib_Manifold_T_Supply : ARRAY[1..GVL_CONSTANTS.C_MAX_MANIFOLDS] OF FB_Sensor_Calibration_Processor;
    fbCalib_Manifold_T_Return : ARRAY[1..GVL_CONSTANTS.C_MAX_MANIFOLDS] OF FB_Sensor_Calibration_Processor;
    fbCalib_Methane : ARRAY[1..GVL_CONSTANTS.C_MAX_METHANE_SENSORS] OF FB_Sensor_Calibration_Processor;
    fbCalib_CO : ARRAY[1..GVL_CONSTANTS.C_MAX_CO_SENSORS] OF FB_Sensor_Calibration_Processor;
    fbAnalog_Manifold_Pressure : ARRAY[1..GVL_CONSTANTS.C_MAX_MANIFOLDS] OF FB_Sensor_Analog_Processing;
    fbAnalog_Manifold_Current : ARRAY[1..GVL_CONSTANTS.C_MAX_MANIFOLDS] OF FB_Sensor_Analog_Processing;
  END_VAR

            // ===== ORIGINAL SNAPSHOT (FULL) =====
fbIO_Watchdog_1(VI_System_Time_MS := GVL_STATUS.G_System_Time_MS, VI_Module_ID := 1, VI_Heartbeat_Signal := GVL_IO.DI_Module_1_Heartbeat, VI_Timeout_MS := 2000);
fbIO_Watchdog_2(VI_System_Time_MS := GVL_STATUS.G_System_Time_MS, VI_Module_ID := 2, VI_Heartbeat_Signal := GVL_IO.DI_Module_2_Heartbeat, VI_Timeout_MS := 2000);

GVL_STATUS.G_IO_Modules_Online[1] := fbIO_Watchdog_1.VO_Module_Online;
GVL_STATUS.G_IO_Modules_Online[2] := fbIO_Watchdog_2.VO_Module_Online;

L_IO_Error_Active := fbIO_Watchdog_1.VO_Error_Active OR fbIO_Watchdog_2.VO_Error_Active;

// IO watchdog events
fbDiagEventManager(
    VI_Code := 16#E001,
    VI_Severity := 4,
    VI_Active := NOT fbIO_Watchdog_1.VO_Module_Online,
    VI_Timestamp := GVL_STATUS.G_System_Time_MS,
    VI_Source := 1,
    VIO_Events := GVL_STATUS.G_Diagnostics_Events,
    VIO_Count := GVL_STATUS.G_Diagnostics_Count
);

fbDiagEventManager(
    VI_Code := 16#E002,
    VI_Severity := 4,
    VI_Active := NOT fbIO_Watchdog_2.VO_Module_Online,
    VI_Timestamp := GVL_STATUS.G_System_Time_MS,
    VI_Source := 2,
    VIO_Events := GVL_STATUS.G_Diagnostics_Events,
    VIO_Count := GVL_STATUS.G_Diagnostics_Count
);

IF L_IO_Error_Active THEN
    GVL_COMMAND.G_Gas_Valve_Close := TRUE;
    GVL_COMMAND.G_Close_Valve_35 := TRUE;
    GVL_COMMAND.G_Close_Valve_36 := TRUE;
    FOR L_i := 1 TO GVL_CONSTANTS.C_MAX_MANIFOLDS DO GVL_STATE.G_Manifold_Pumps[L_i] := FALSE; END_FOR;
END_IF;

FOR L_i := 1 TO 8 DO
    fbDebounce_Switches[L_i](IN := GVL_IO.DI_Lighting_Switches[L_i], PT := L_Debounce_Time, VI_System_Time_MS := GVL_STATUS.G_System_Time_MS);
    GVL_STATE.G_Physical_Switches[L_i] := fbDebounce_Switches[L_i].Q;
    
    fbDebounce_Motion[L_i](IN := GVL_IO.DI_Motion_Sensors[L_i], PT := L_Debounce_Time, VI_System_Time_MS := GVL_STATUS.G_System_Time_MS);
    GVL_STATE.G_Motion_Sensors[L_i] := fbDebounce_Motion[L_i].Q;
END_FOR;

FOR L_i := 1 TO GVL_CONSTANTS.C_MAX_SOCKETS DO
    GVL_STATE.G_Socket_Switches[L_i] := FALSE;
END_FOR;

FOR L_i := 1 TO GVL_CONSTANTS.C_MAX_SECURITY_SENSORS DO
    fbDebounce_Security_Open[L_i](IN := GVL_IO.DI_Security_Open[L_i], PT := L_Debounce_Time, VI_System_Time_MS := GVL_STATUS.G_System_Time_MS);
    fbDebounce_Security_Glass[L_i](IN := GVL_IO.DI_Security_Glass[L_i], PT := L_Debounce_Time, VI_System_Time_MS := GVL_STATUS.G_System_Time_MS);
END_FOR;

fbDebounce_Group_2F(IN := GVL_IO.DI_Security_2F_Group, PT := L_Debounce_Time, VI_System_Time_MS := GVL_STATUS.G_System_Time_MS);

FOR L_i := 1 TO GVL_CONSTANTS.C_MAX_DOOR_SENSORS DO
    IF GVL_CONFIG.G_Door_Map[L_i] > 0 AND GVL_CONFIG.G_Door_Map[L_i] <= GVL_CONSTANTS.C_MAX_SECURITY_SENSORS THEN
        GVL_STATE.G_Door_Sensors[L_i] := fbDebounce_Security_Open[GVL_CONFIG.G_Door_Map[L_i]].Q;
    END_IF;
END_FOR;

FOR L_i := 1 TO 8 DO
    IF GVL_CONFIG.G_Window_Map[L_i] > 0 THEN
        IF GVL_CONFIG.G_Window_Map[L_i] <= GVL_CONSTANTS.C_MAX_SECURITY_SENSORS THEN
            GVL_STATE.G_Window_Sensors[L_i] := fbDebounce_Security_Open[GVL_CONFIG.G_Window_Map[L_i]].Q;
        ELSE
            GVL_STATE.G_Window_Sensors[L_i] := fbDebounce_Security_Glass[GVL_CONFIG.G_Window_Map[L_i] - GVL_CONSTANTS.C_MAX_SECURITY_SENSORS].Q;
        END_IF;
    END_IF;
END_FOR;
GVL_STATE.G_Window_Sensors[16] := fbDebounce_Group_2F.Q;

FOR L_i := 1 TO GVL_CONSTANTS.C_MAX_FLOOD_SENSORS DO
    fbDebounce_Flood[L_i](IN := GVL_IO.DI_Flood_Sensors[L_i], PT := L_Debounce_Time, VI_System_Time_MS := GVL_STATUS.G_System_Time_MS);
    GVL_STATE.G_Water_Sensors[L_i] := fbDebounce_Flood[L_i].Q;
END_FOR;

FOR L_i := 1 TO GVL_CONSTANTS.C_MAX_SMOKE_SENSORS DO
    fbDebounce_Smoke[L_i](IN := GVL_IO.DI_Smoke_Sensors[L_i], PT := L_Debounce_Time, VI_System_Time_MS := GVL_STATUS.G_System_Time_MS);
    GVL_STATE.G_Smoke_Sensors[L_i] := fbDebounce_Smoke[L_i].Q;
END_FOR;

// ===== ENHANCED LAYER =====
fbCalib_Outdoor_Temp(
    VI_Raw_Value := GVL_IO.AI_Temp_Outdoor.rValue,
    VI_Record := GVL_CONFIG.G_Calib_Outdoor_Temp
);
GVL_STATE.G_Outdoor_Temp := fbCalib_Outdoor_Temp.VO_Calibrated_Value;

FOR L_i := 1 TO GVL_CONSTANTS.C_MAX_SUPPLY_TEMPS DO
    IF GVL_IO.AI_Supply_Temps[L_i].wStatus = 0 THEN
        fbCalib_Supply_Temps[L_i](
            VI_Raw_Value := GVL_IO.AI_Supply_Temps[L_i].rValue,
            VI_Record := GVL_CONFIG.G_Calib_Supply_Temps[L_i]
        );
        GVL_STATE.G_Supply_Temps[L_i] := fbCalib_Supply_Temps[L_i].VO_Calibrated_Value;
    END_IF;
END_FOR;

FOR L_i := 1 TO 8 DO
    fbCalib_Room_Hum[L_i](
        VI_Raw_Value := GVL_IO.AI_Room_Hum[L_i],
        VI_Record := GVL_CONFIG.G_Calib_Humidity[L_i]
    );
    GVL_STATE.G_Room_Hum[L_i] := fbCalib_Room_Hum[L_i].VO_Calibrated_Value;

    fbCalib_Room_CO2[L_i](
        VI_Raw_Value := GVL_IO.AI_Room_CO2[L_i],
        VI_Record := GVL_CONFIG.G_Calib_CO2[L_i]
    );
    GVL_STATE.G_Room_CO2[L_i] := fbCalib_Room_CO2[L_i].VO_Calibrated_Value;
END_FOR;

FOR L_i := 1 TO 8 DO
    fbCalib_Room_Temps[L_i](
        VI_Raw_Value := GVL_IO.AI_Room_Temps[L_i],
        VI_Record := GVL_CONFIG.G_Calib_Room_Temps[L_i]
    );
    GVL_STATE.G_Room_Temps[L_i] := fbCalib_Room_Temps[L_i].VO_Calibrated_Value;

    fbCalib_Floor_Temps[L_i](
        VI_Raw_Value := GVL_IO.AI_Floor_Temps[L_i],
        VI_Record := GVL_CONFIG.G_Calib_Floor_Temps[L_i]
    );
    GVL_STATE.G_Floor_Temps[L_i] := fbCalib_Floor_Temps[L_i].VO_Calibrated_Value;
END_FOR;

GVL_STATUS.G_Diagnostics.Manifold_Pressure_Fault_Active := FALSE;
GVL_STATUS.G_Diagnostics.Manifold_Pressure_First_Fault_Index := 0;
GVL_STATUS.G_Diagnostics.Manifold_Current_Fault_Active := FALSE;
GVL_STATUS.G_Diagnostics.Manifold_Current_First_Fault_Index := 0;
GVL_STATUS.G_Diagnostics.Manifold_Pressure_Fault_Text := '';
GVL_STATUS.G_Diagnostics.Manifold_Current_Fault_Text := '';
GVL_STATUS.G_Diagnostics.Sensor_Fault := FALSE;
GVL_STATUS.G_Diagnostics.Subsystem_Degraded := FALSE;

FOR L_i := 1 TO GVL_CONSTANTS.C_MAX_MANIFOLDS DO
    IF GVL_IO.AI_Manifold_Pressures[L_i] < 0 THEN
        L_Manifold_Pressure_Raw := 0;
    ELSE
        L_Manifold_Pressure_Raw := INT_TO_WORD(GVL_IO.AI_Manifold_Pressures[L_i]);
    END_IF;

    IF GVL_IO.AI_Manifold_Currents[L_i] < 0 THEN
        L_Manifold_Current_Raw := 0;
    ELSE
        L_Manifold_Current_Raw := INT_TO_WORD(GVL_IO.AI_Manifold_Currents[L_i]);
    END_IF;

    fbAnalog_Manifold_Pressure[L_i](
        VI_Raw_Value := L_Manifold_Pressure_Raw,
        VI_Sensor_Type := 0,
        VI_Min_Scale := 0.0,
        VI_Max_Scale := 10.0,
        VI_Offset := 0.0,
        VI_Multiplier := 1.0,
        VI_Filter_Time_MS := GVL_CONSTANTS.C_MS_IN_SECOND,
        VI_System_Time_MS := GVL_STATUS.G_System_Time_MS,
        VI_Fallback_Mode := 0,
        VI_Default_Value := 0.0
    );
    GVL_STATE.G_Manifold_Pressures[L_i] := fbAnalog_Manifold_Pressure[L_i].VO_Value;
    GVL_STATUS.G_Diagnostics.Manifold_Pressure_Fault[L_i] := fbAnalog_Manifold_Pressure[L_i].VO_Error;
    GVL_STATUS.G_Diagnostics.Manifold_Pressure_Diag_Code[L_i] := fbAnalog_Manifold_Pressure[L_i].VO_Diag_Code;

    fbDiagEventManager(
        VI_Code := GVL_CONFIG.ERR_PRESSURE_OUT_OF_RANGE,
        VI_Severity := 3,
        VI_Active := fbAnalog_Manifold_Pressure[L_i].VO_Error,
        VI_Timestamp := GVL_STATUS.G_System_Time_MS,
        VI_Source := 100 + L_i,
        VIO_Events := GVL_STATUS.G_Diagnostics_Events,
        VIO_Count := GVL_STATUS.G_Diagnostics_Count
    );

    fbAnalog_Manifold_Current[L_i](
        VI_Raw_Value := L_Manifold_Current_Raw,
        VI_Sensor_Type := 0,
        VI_Min_Scale := 0.0,
        VI_Max_Scale := 16.0,
        VI_Offset := 0.0,
        VI_Multiplier := 1.0,
        VI_Filter_Time_MS := GVL_CONSTANTS.C_MS_IN_SECOND,
        VI_System_Time_MS := GVL_STATUS.G_System_Time_MS,
        VI_Fallback_Mode := 0,
        VI_Default_Value := 0.0
    );
    GVL_STATE.G_Manifold_Currents[L_i] := fbAnalog_Manifold_Current[L_i].VO_Value;
    GVL_STATUS.G_Diagnostics.Manifold_Current_Fault[L_i] := fbAnalog_Manifold_Current[L_i].VO_Error;
    GVL_STATUS.G_Diagnostics.Manifold_Current_Diag_Code[L_i] := fbAnalog_Manifold_Current[L_i].VO_Diag_Code;

    fbDiagEventManager(
        VI_Code := GVL_CONFIG.ERR_PUMP_UNDERCURRENT,
        VI_Severity := 3,
        VI_Active := fbAnalog_Manifold_Current[L_i].VO_Error,
        VI_Timestamp := GVL_STATUS.G_System_Time_MS,
        VI_Source := 200 + L_i,
        VIO_Events := GVL_STATUS.G_Diagnostics_Events,
        VIO_Count := GVL_STATUS.G_Diagnostics_Count
    );

    IF GVL_IO.AI_Manifold_Temps_Supply[L_i].wStatus = 0 THEN
        fbCalib_Manifold_T_Supply[L_i](
            VI_Raw_Value := GVL_IO.AI_Manifold_Temps_Supply[L_i].rValue,
            VI_Record := GVL_CONFIG.G_Calib_Manifold_T_Supply[L_i]
        );
        GVL_STATE.G_Manifold_T_Supply[L_i] := fbCalib_Manifold_T_Supply[L_i].VO_Calibrated_Value;
    END_IF;

    fbCalib_Manifold_T_Return[L_i](
        VI_Raw_Value := INT_TO_REAL(GVL_IO.AI_Manifold_Temps_Return[L_i]) / 10.0,
        VI_Record := GVL_CONFIG.G_Calib_Manifold_T_Return[L_i]
    );
    GVL_STATE.G_Manifold_T_Return[L_i] := fbCalib_Manifold_T_Return[L_i].VO_Calibrated_Value;
    GVL_STATE.G_Manifold_End_Switches[L_i] := GVL_IO.DI_Manifold_End_Switches[L_i];

    IF GVL_STATUS.G_Diagnostics.Manifold_Pressure_Fault[L_i] OR GVL_STATUS.G_Diagnostics.Manifold_Current_Fault[L_i] THEN
        GVL_STATUS.G_Diagnostics.Sensor_Fault := TRUE;
        GVL_STATUS.G_Diagnostics.Subsystem_Degraded := TRUE;
    END_IF;

    IF GVL_STATUS.G_Diagnostics.Manifold_Pressure_Fault[L_i] AND GVL_STATUS.G_Diagnostics.Manifold_Current_Fault[L_i] THEN
        GVL_STATUS.G_Diagnostics.Manifold_Pressure_Fault_Text := 'Correlated pressure/current fault detected';
        GVL_STATUS.G_Diagnostics.Manifold_Current_Fault_Text := 'Correlated pressure/current fault detected';
    ELSIF GVL_STATUS.G_Diagnostics.Manifold_Pressure_Fault[L_i] AND (GVL_STATUS.G_Diagnostics.Manifold_Pressure_Fault_Text = '') THEN
        GVL_STATUS.G_Diagnostics.Manifold_Pressure_Fault_Text := 'Pressure sensor fault detected';
    ELSIF GVL_STATUS.G_Diagnostics.Manifold_Current_Fault[L_i] AND (GVL_STATUS.G_Diagnostics.Manifold_Current_Fault_Text = '') THEN
        GVL_STATUS.G_Diagnostics.Manifold_Current_Fault_Text := 'Current sensor fault detected';
    END_IF;
END_FOR;

FOR L_i := 1 TO GVL_CONSTANTS.C_MAX_METHANE_SENSORS DO
    IF GVL_IO.AI_Methane_LEL[L_i].wStatus = 0 THEN
        fbCalib_Methane[L_i](
            VI_Raw_Value := GVL_IO.AI_Methane_LEL[L_i].rValue,
            VI_Record := GVL_CONFIG.G_Calib_Methane[L_i]
        );
        GVL_STATE.G_Methane_Sensors[L_i] := fbCalib_Methane[L_i].VO_Calibrated_Value;
    END_IF;

    fbDiagEventManager(
        VI_Code := 16#E003,
        VI_Severity := 3,
        VI_Active := GVL_IO.AI_Methane_LEL[L_i].wStatus <> 0,
        VI_Timestamp := GVL_STATUS.G_System_Time_MS,
        VI_Source := 300 + L_i,
        VIO_Events := GVL_STATUS.G_Diagnostics_Events,
        VIO_Count := GVL_STATUS.G_Diagnostics_Count
    );
END_FOR;

FOR L_i := 1 TO GVL_CONSTANTS.C_MAX_CO_SENSORS DO
    fbCalib_CO[L_i](
        VI_Raw_Value := GVL_IO.AI_CO_PPM[L_i],
        VI_Record := GVL_CONFIG.G_Calib_CO[L_i]
    );
    GVL_STATE.G_CO_Sensors[L_i] := fbCalib_CO[L_i].VO_Calibrated_Value;
END_FOR;

GVL_STATE.G_Boiler_Flame := GVL_IO.AI_Boiler_Flame_Status;
GVL_STATE.G_Boiler_Error := GVL_IO.DI_Boiler_Error;
FOR L_i := 1 TO GVL_CONSTANTS.C_MAX_BOILERS DO
    GVL_STATE.G_Boiler_OT_Online[L_i] := FALSE;
END_FOR;

GVL_STATE.G_DHW_Temp := GVL_IO.AI_DHW_Temp;
GVL_STATE.G_DHW_Pressure := GVL_IO.AI_DHW_Pressure;

GVL_STATE.G_Water_Zone_Open_FB := GVL_IO.DI_Water_Zone_Open_FB;
GVL_STATE.G_Water_Zone_Close_FB := GVL_IO.DI_Water_Zone_Close_FB;

// >>> BULK_SYNC_ANCHOR: PRG_IO_Read <<<
          
END_PROGRAM

PROGRAM PRG_PLC_B

            // Вызов основной программы
PRG_System();
// >>> BULK_SYNC_ANCHOR: PRG_PLC_B <<<
          
END_PROGRAM

PROGRAM PRG_Ventilation
  VAR
    fbVentilationManager : FB_Ventilation_System_Manager;
    L_i : INT;
    L_Supply_Fans_Byte : ARRAY[1..GVL_CONSTANTS.C_MAX_SUPPLY_FANS] OF BYTE;
    L_Exhaust_Fans_Byte : ARRAY[1..GVL_CONSTANTS.C_MAX_EXHAUST_FANS] OF BYTE;
    L_Wet_Zone_Active : ARRAY[1..GVL_CONSTANTS.C_MAX_WET_ZONES] OF BOOL;
    L_Vent_PV3_Boost_Req : BOOL;
    L_Supply_100_Req : BOOL;
    L_Exhaust_100_Req : BOOL;
    L_Supply_80_Req : BOOL;
    L_Vent_Stop_Req : BOOL;
  END_VAR

            // Wet-zone adapter
FOR L_i := 1 TO GVL_CONSTANTS.C_MAX_WET_ZONES DO
    L_Wet_Zone_Active[L_i] := FALSE;
END_FOR;
IF GVL_STATUS.G_Wet_Zone_Light_Active THEN
    L_Wet_Zone_Active[1] := TRUE;
END_IF;

// === Ventilation Inputs (from arbitration only) ===
L_Vent_PV3_Boost_Req := GVL_COMMAND_SHADOW.G_Vent_PV3_Boost;
L_Supply_100_Req := GVL_COMMAND_SHADOW.G_Supply_100_Req;
L_Exhaust_100_Req := GVL_COMMAND_SHADOW.G_Exhaust_100_Req;
L_Supply_80_Req := GVL_COMMAND_SHADOW.G_Supply_80_Req;
L_Vent_Stop_Req := GVL_COMMAND_SHADOW.G_Vent_Stop;

// Coordinator constraint: block non-stop ventilation requests only.
// Safety-driven stop request must remain untouched.
IF GVL_SYSTEM_COORDINATION.G_Block_Ventilation THEN
    L_Vent_PV3_Boost_Req := FALSE;
    L_Supply_100_Req := FALSE;
    L_Exhaust_100_Req := FALSE;
    L_Supply_80_Req := FALSE;
END_IF;

// 11. Управление вентиляцией
fbVentilationManager(
    VI_System_Time_MS := GVL_STATUS.G_System_Time_MS,
    VI_IsActivePLC := GVL_STATUS.G_Is_Active_PLC,
    VI_Outdoor_Temp := GVL_STATE.G_Outdoor_Temp,
    VI_Supply_Temps := GVL_STATE.G_Supply_Temps,
    VI_Room_Temps := GVL_STATE.G_Room_Temps,
    VI_Room_Humidities := GVL_STATE.G_Room_Hum,
    VI_Room_CO2 := GVL_STATE.G_Room_CO2,
    VI_Current_Scenario := GVL_STATUS.G_Current_Scenario,
    VI_System_Mode := GVL_STATE.G_System_Mode,
    VI_Config := GVL_CONFIG.G_HMI_Vent_Global_Config,
    VI_Fire_Alarm := GVL_STATE.G_Safety_Smoke_Latched,
    VI_Gas_Alarm := GVL_STATE.G_Safety_Gas_Latched,
    VI_PV3_Boost_Req := L_Vent_PV3_Boost_Req,
    VI_Supply_100_Req := L_Supply_100_Req,
    VI_Exhaust_100_Req := L_Exhaust_100_Req,
    VI_Supply_80_Req := L_Supply_80_Req,
    VI_Vent_Stop := L_Vent_Stop_Req,
    VI_IO_Modules_Online := GVL_STATUS.G_IO_Modules_Online,
    VI_Wet_Zone_Active := L_Wet_Zone_Active,
    VI_Rule_Actions := GVL_STATE.G_Rule_Actions,
    VO_Supply_Fans => L_Supply_Fans_Byte,
    VO_Exhaust_Fans => L_Exhaust_Fans_Byte,
    VO_Heater_Power => GVL_STATE.G_Vent_Heater_Power,
    VO_Status_Msg => GVL_STATUS.G_Vent_Status_Msg,
    VO_Ventilation_IO_Fault => GVL_STATE.G_Ventilation_IO_Fault,
    VO_Ventilation_Subsystem_Degraded => GVL_STATE.G_Ventilation_Subsystem_Degraded
);
// >>> BULK_SYNC_ANCHOR: PRG_Ventilation <<<


// Ventilation copy-out adapters
FOR L_i := 1 TO GVL_CONSTANTS.C_MAX_SUPPLY_FANS DO
    GVL_STATE.G_Supply_Fans[L_i] := BYTE_TO_REAL(L_Supply_Fans_Byte[L_i]);
END_FOR;
FOR L_i := 1 TO GVL_CONSTANTS.C_MAX_EXHAUST_FANS DO
    GVL_STATE.G_Exhaust_Fans[L_i] := BYTE_TO_REAL(L_Exhaust_Fans_Byte[L_i]);
END_FOR;
          
END_PROGRAM

PROGRAM PRG_System
  VAR
    L_i : INT;
    L_Motion_Sensors_16 : ARRAY[1..16] OF BOOL;
    L_Zone_Valves_8 : ARRAY[1..8] OF BOOL;
    L_Lighting_32 : ARRAY[1..32] OF BYTE;
    L_Lighting_Bool_32 : ARRAY[1..32] OF BOOL;
    L_FloorTemps_8 : ARRAY[1..8] OF REAL;
    fbCoreKernelObserver : FB_CoreKernel_Live_Observer;    fbSimulationManager : FB_Simulation_Manager;
    fbRuleEngine : FB_Rule_Engine;
    fbBlackBox : FB_BlackBox_Recorder;
    fbAstroTimer : FB_Astro_Timer;    fbHistoryManager : FB_History_Manager;    fbLogEvent : FB_LogEvent;
    fbSystemScenarioArb : FB_System_Scenario_Arbitration;
    fbSystemGatewayIntent : FB_System_Gateway_Intent;
    fbSystemPersist : FB_System_Persist_Manager;
    fbSystemInit : FB_System_Init;
    fbSystemRecovery : FB_System_Recovery;
    fbTimebase : FB_System_Timebase;
    fbSystemRedundancy : FB_System_Redundancy_Orchestrator;
    fbSystemHealthOrchestrator : FB_System_Health_Orchestrator;
    fbSystemIntentPublisher : FB_System_Intent_Publisher;
    fbSystemEvacuation : FB_System_Evacuation;
    fbSystemAlarmOrchestrator : FB_System_Alarm_Orchestrator;
    L_Time_Diff : UDINT;
    L_Local_State : ST_System_State_Snapshot;
    L_Remote_State : ST_System_State_Snapshot;
    L_NVRAM_Cmd : BYTE;
    L_NVRAM_Offset : UDINT;
    L_NVRAM_Done : BOOL;
    L_NVRAM_Err : BOOL;
    L_NVRAM_ErrID : UDINT;
    L_BB_Record : ST_BlackBox_Record;
    L_BB_Freeze : BOOL;
    L_Scenario_Idx : INT;
    L_Last_Operator_Blocked : BOOL;
    L_Last_DHW_Heating_In_Service : BOOL;
    L_Last_DHW_Circ_In_Service : BOOL;
    L_Dangerous_Action_Armed : BOOL;
    L_Dangerous_Action_Deadline_MS : UDINT;
    L_Maintenance_Apply_Intent : BOOL;
    L_Last_System_Mode : E_System_Operating_Mode;
    L_Last_First_Fault_Type : INT;
    L_Last_First_Fault_Source : INT;
    L_First_Fault_Active : BOOL;
    L_First_Fault_Type : INT;
    L_First_Fault_Source : INT;
    L_System_Severity : E_System_Severity;
    L_Root_Cause : E_System_Root_Cause;
    L_Watchdog_Fault : BOOL;
    L_Last_Root_Cause : E_System_Root_Cause;
    L_History_Event : ST_History_Record;
    L_History_Write_Event : BOOL;
    L_Last_Operator_Journal_Seq : UDINT;
    L_Last_Event_Code : UDINT;
    L_Last_Event_Value : REAL;
    L_Last_Event_Time_MS : UDINT;
    L_Gateway_Writes_Allowed : BOOL;
    L_Scenario_Req_Operator : E_SCENARIO_TYPE;
    L_Scenario_Req_Gateway : E_SCENARIO_TYPE;
    L_Scenario_Req_Rule : E_SCENARIO_TYPE;
    L_Scenario_Req_Final : E_SCENARIO_TYPE;
    L_Scenario_Intent : E_SCENARIO_TYPE;
    L_Scenario_Source : E_SCENARIO_SOURCE;
    L_Scenario_Changed : BOOL;
    L_Last_Scenario_Change_Time : UDINT;
    L_IO_Fault : BOOL;
    L_IO_Fault_Prev : BOOL;
    L_Comm_Fault_Prev : BOOL;
    L_Sensor_Fault_Prev : BOOL;
    L_Subsystem_Fault_Prev : BOOL;
    L_Mode_Prev : E_System_Operating_Mode;
    L_User_Access_Denied_Prev : BOOL;
    L_Persist_Buffer : ARRAY[0..4] OF BYTE;
    L_Last_Written_Persist_Buffer : ARRAY[0..4] OF BYTE;
    L_Persist_Buffer_Changed : BOOL;
    L_Last_Persist_Write_MS : UDINT;
    L_Recovery_Done : BOOL;
    L_Persist_Struct : ST_Persist;
  END_VAR

            // 0. Инициализация RETAIN переменных при первом запуске
fbSystemInit(
    VIO_Local_State := L_Local_State,
    VIO_Remote_State := L_Remote_State
);

// === NVRAM RECOVERY (ONCE AFTER BOOT) ===
fbSystemRecovery(
    VIO_Recovery_Done := L_Recovery_Done
);

// === Persist manager ===
fbSystemPersist(
    VI_System_Time_MS := GVL_STATUS.G_System_Time_MS,
    VI_IsActivePLC := GVL_STATUS.G_Is_Active_PLC,
    VIO_Persist_Buffer := L_Persist_Buffer,
    VIO_Last_Written_Persist_Buffer := L_Last_Written_Persist_Buffer,
    VIO_Persist_Buffer_Changed := L_Persist_Buffer_Changed,
    VIO_Last_Persist_Write_MS := L_Last_Persist_Write_MS,
    VIO_NVRAM_Cmd := L_NVRAM_Cmd,
    VIO_NVRAM_Offset := L_NVRAM_Offset,
    VIO_NVRAM_Done := L_NVRAM_Done,
    VIO_NVRAM_Err := L_NVRAM_Err,
    VIO_NVRAM_ErrID := L_NVRAM_ErrID
);

// NVRAM CONTROLLED WRITE ENABLED (step 8B)

// 1. Обновление системного времени
fbTimebase();

// 2-3. Redundancy / state sync
fbSystemRedundancy(
    VIO_Local_State := L_Local_State,
    VIO_Remote_State := L_Remote_State
);

// 3.4-3.7. Safety / health / state mode
fbSystemHealthOrchestrator(
    VO_First_Fault_Active => L_First_Fault_Active,
    VO_First_Fault_Type => L_First_Fault_Type,
    VO_First_Fault_Source => L_First_Fault_Source,
    VO_System_Severity => L_System_Severity,
    VO_Root_Cause => L_Root_Cause,
    VO_Watchdog_Fault => L_Watchdog_Fault
);

// === STAGE G2b: SYSTEM GATE PUBLICATION ===
fbSystemIntentPublisher(
    VI_System_Time_MS := GVL_STATUS.G_System_Time_MS,
    VI_Gateway_Writes_Allowed := L_Gateway_Writes_Allowed
);

// 3.6a. Эвакуация
fbSystemEvacuation();

// 4. Астрономический таймер
fbAstroTimer(
    VI_System_Time_MS := GVL_STATUS.G_System_Time_MS,
    VI_Latitude := 55.75,
    VI_Longitude := 37.61,
    VI_Day_Of_Year := GVL_STATUS.G_Day_Of_Year,
    VO_Is_Night => GVL_STATUS.G_Is_Night
);


// 5. Управление сценариями
// Scenario request (direct + early operator gate)
IF GVL_STATE.G_System_Mode = E_System_Operating_Mode.MODE_NORMAL THEN
    L_Scenario_Req_Operator := GVL_COMMAND.G_Scenario_Request_Operator;
ELSE
    L_Scenario_Req_Operator := E_SCENARIO_TYPE.SCENARIO_NONE;
END_IF;
L_Scenario_Req_Gateway := 0;
L_Scenario_Req_Rule := 0;







// Синхронизируем request с фактически активным сценарием


L_Scenario_Idx := TO_INT(GVL_STATUS.G_Current_Scenario);
IF L_Scenario_Idx < 0 OR L_Scenario_Idx > 7 THEN
    L_Scenario_Idx := 0;
END_IF;

// === Scenario arbitration ===
fbSystemScenarioArb(
    VI_System_Time_MS := GVL_STATUS.G_System_Time_MS,
    VI_IsActivePLC := GVL_STATUS.G_Is_Active_PLC,
    VI_System_Mode := GVL_STATE.G_System_Mode,
    VI_Security_Armed := GVL_ALARM.G_Security_Armed,
    VIO_Scenario_Req_Operator := L_Scenario_Req_Operator,
    VIO_Scenario_Req_Gateway := L_Scenario_Req_Gateway,
    VIO_Scenario_Req_Rule := L_Scenario_Req_Rule,
    VIO_Scenario_Req_Final := L_Scenario_Req_Final,
    VIO_Scenario_Intent := L_Scenario_Intent,
    VIO_Scenario_Source := L_Scenario_Source
);

// 6. Симуляция присутствия
fbSimulationManager(
    VI_System_Time_MS := GVL_STATUS.G_System_Time_MS,
    VI_IsActivePLC := GVL_STATUS.G_Is_Active_PLC AND (GVL_STATE.G_System_Mode = E_System_Operating_Mode.MODE_NORMAL),
    VI_Scenario := GVL_STATUS.G_Current_Scenario,
    VI_Config := GVL_CONFIG.G_HMI_Scenario_Configs[L_Scenario_Idx],
    VO_Sim_Lights => GVL_STATE.G_Sim_Lights,
    VO_Sim_Active => GVL_STATUS.G_Sim_Active
);

// 6.5. Пользовательские правила (Rule Engine)
fbRuleEngine(
    VI_System_Time_MS := GVL_STATUS.G_System_Time_MS,
    VI_IsActivePLC := GVL_STATUS.G_Is_Active_PLC,
    VI_Rules := GVL_CONFIG.G_HMI_User_Rules,
    VI_Indoor_Temps := GVL_STATE.G_Room_Temps,
    VI_Floor_Temps := L_FloorTemps_8,
    VI_Humidities := GVL_STATE.G_Room_Hum,
    VI_CO2_Levels := GVL_STATE.G_Room_CO2,
    VI_Motion_Sensors := L_Motion_Sensors_16,
    VI_Door_Sensors := GVL_STATE.G_Door_Sensors,
    VI_Window_Sensors := GVL_STATE.G_Window_Sensors,
    VI_Water_Sensors := GVL_STATE.G_Water_Sensors,
    VI_Smoke_Sensors := GVL_STATE.G_Smoke_Sensors,
    VI_Methane_Sensors := GVL_STATE.G_Methane_Sensors,
    VI_CO_Sensors := GVL_STATE.G_CO_Sensors,
    VI_Security_Armed := GVL_ALARM.G_Security_Armed,
    VI_Current_Time := GVL_STATUS.G_Current_TOD,
    VI_Day_Of_Week := TO_INT(GVL_STATUS.G_Current_Day),
    VO_Actions => GVL_STATE.G_Rule_Actions
);

FOR L_i := 1 TO GVL_CONSTANTS.C_MAX_RULES DO
    IF GVL_STATE.G_Rule_Actions[L_i].Active AND GVL_STATE.G_Rule_Actions[L_i].Action_Type = E_Rule_Action_Type.ACTION_ACTIVATE_SCENARIO THEN
        L_Scenario_Req_Rule := TO_BYTE(GVL_STATE.G_Rule_Actions[L_i].Value);
    END_IF;
END_FOR;



// 8.5 Менеджер тревог
fbSystemAlarmOrchestrator(
    VI_First_Fault_Active := L_First_Fault_Active,
    VI_First_Fault_Type := L_First_Fault_Type,
    VI_First_Fault_Source := L_First_Fault_Source
);

// Command arbitration: OPERATOR > GATEWAY
L_Gateway_Writes_Allowed :=
    NOT GVL_STATUS.G_Diagnostics.Dangerous_Action_Pending_Confirm AND
    NOT GVL_STATUS.G_Diagnostics.Operator_Action_Blocked AND
    NOT GVL_STATUS.G_Diagnostics.User_Access_Denied;

// === Gateway intent ===
fbSystemGatewayIntent(
    VI_System_Time_MS := GVL_STATUS.G_System_Time_MS,
    VI_IsActivePLC := GVL_STATUS.G_Is_Active_PLC,
    VI_Gateway_Writes_Allowed := L_Gateway_Writes_Allowed,
    VIO_FloorHeating_Temps := L_FloorTemps_8,
    VIO_Zone_Valve_States := L_Zone_Valves_8,
    VIO_Lighting_Base_Levels := L_Lighting_32,
    VIO_Scenario_Req_Gateway := L_Scenario_Req_Gateway
);

// Gateway moved to helper

// Persist/NVRAM moved to helper

// 15. Черный ящик
L_BB_Record.Timestamp := GVL_STATUS.G_System_Time_MS;
L_BB_Record.PLC_Active_ID := GVL_STATUS.G_PLC_ID;
L_BB_Record.Gas_Methane_LEL := GVL_STATE.G_Methane_Sensors[1];
L_BB_Record.Gas_CO_PPM := GVL_STATE.G_CO_Sensors[1];
L_BB_Record.Flood_Active := GVL_ALARM.G_Flood_Alarm_Active;
L_BB_Record.Fire_Active := GVL_ALARM.G_Fire_Alarm_Active;
L_BB_Record.Valve_Gas_Status := SEL(GVL_COMMAND.G_Gas_Valve_Close, BYTE#0, BYTE#1);
L_BB_Record.Valve_Water_Status := SEL((GVL_COMMAND.G_Close_Valve_35 OR GVL_COMMAND.G_Close_Valve_36), BYTE#0, BYTE#1);

L_BB_Record.System_Mode := TO_BYTE(TO_INT(GVL_STATE.G_System_Mode));
L_BB_Record.First_Fault_Type := TO_BYTE(TO_INT(L_First_Fault_Type));
L_BB_Record.First_Fault_Source := TO_BYTE(TO_INT(L_First_Fault_Source));
L_BB_Record.First_Fault_Active := L_First_Fault_Active;
L_BB_Record.System_Severity := TO_BYTE(TO_INT(L_System_Severity));
L_BB_Record.Root_Cause := TO_BYTE(TO_INT(L_Root_Cause));
L_BB_Record.Watchdog_Fault := L_Watchdog_Fault;


L_BB_Freeze := GVL_ALARM.G_Gas_Alarm_Active OR GVL_ALARM.G_Fire_Alarm_Active OR GVL_ALARM.G_Flood_Alarm_Active OR L_First_Fault_Active;

fbBlackBox(
    VI_Current_Data := L_BB_Record,
    VI_Freeze := L_BB_Freeze
);

// 15.1. Менеджер истории / diagnostics bridge
L_History_Write_Event := FALSE;
L_History_Event.timestamp_ms := GVL_STATUS.G_System_Time_MS;
L_History_Event.event_code := 0;
L_History_Event.event_value := 0.0;
L_History_Event.unit := 0;
L_History_Event.zone_id := 0;
L_History_Event.operator_id := 'SYSTEM';
L_History_Event.priority := E_ALERT_PRIORITY.ALERT_PRIORITY_HIGH;

IF GVL_STATE.G_System_Mode <> L_Last_System_Mode THEN
    L_History_Write_Event := TRUE;
    L_History_Event.event_code := 1101; // System mode transition
    L_History_Event.event_value := TO_REAL(TO_INT(GVL_STATE.G_System_Mode));
    L_History_Event.unit := 1; // system mode domain
    L_History_Event.zone_id := 0;
    IF GVL_STATE.G_System_Mode = E_System_Operating_Mode.MODE_NORMAL THEN
        L_History_Event.priority := E_ALERT_PRIORITY.ALERT_PRIORITY_HIGH;
    ELSE
        L_History_Event.priority := E_ALERT_PRIORITY.ALERT_PRIORITY_HIGH;
    END_IF;
    L_Last_System_Mode := GVL_STATE.G_System_Mode;

ELSIF L_Root_Cause <> L_Last_Root_Cause THEN
    L_History_Write_Event := TRUE;
    L_History_Event.event_code := 1102; // Root cause changed
    L_History_Event.event_value := TO_REAL(TO_INT(L_Root_Cause));
    L_History_Event.unit := 2; // root cause enum domain
    L_History_Event.zone_id := TO_BYTE(L_First_Fault_Source);
    L_History_Event.priority := E_ALERT_PRIORITY.ALERT_PRIORITY_HIGH;
    L_Last_Root_Cause := L_Root_Cause;

ELSIF L_First_Fault_Source <> L_Last_First_Fault_Source THEN
    L_History_Write_Event := TRUE;
    L_History_Event.event_code := 1103; // First fault source changed
    L_History_Event.event_value := TO_REAL(L_First_Fault_Source);
    L_History_Event.unit := 3; // root cause source domain
    L_History_Event.zone_id := TO_BYTE(L_First_Fault_Source);
    L_History_Event.priority := E_ALERT_PRIORITY.ALERT_PRIORITY_HIGH;
    L_Last_First_Fault_Source := L_First_Fault_Source;

ELSIF GVL_STATUS.G_Current_Scenario <> GVL_STATUS.G_Previous_Scenario THEN
    L_History_Write_Event := TRUE;
    L_History_Event.event_code := 1001; // Scenario transition
    L_History_Event.event_value := TO_REAL(GVL_STATUS.G_Current_Scenario);
    L_History_Event.unit := 4; // scenario domain
    L_History_Event.zone_id := 0;
    L_History_Event.priority := E_ALERT_PRIORITY.ALERT_PRIORITY_HIGH;
    GVL_STATUS.G_Previous_Scenario := GVL_STATUS.G_Current_Scenario;

ELSIF GVL_STATUS.G_Diagnostics.Alarm_Event_Pulse THEN
    L_History_Write_Event := TRUE;
    L_History_Event.event_code := TO_WORD(GVL_STATUS.G_Diagnostics.Alarm_Event_Code);
    L_History_Event.event_value := GVL_STATUS.G_Diagnostics.Alarm_Event_Value;
    L_History_Event.unit := 10; // alarm lifecycle domain
    L_History_Event.zone_id := 0;
    L_History_Event.priority := E_ALERT_PRIORITY.ALERT_PRIORITY_HIGH;

ELSIF GVL_STATUS.G_Diagnostics.Operator_Journal_Event_Seq <> L_Last_Operator_Journal_Seq THEN
    L_History_Write_Event := TRUE;
    L_History_Event.event_code := 1301; // Operator journal event
    L_History_Event.event_value := TO_REAL(GVL_STATUS.G_Diagnostics.Operator_Journal_Event_Seq);
    L_History_Event.unit := 20; // operator journal domain
    L_History_Event.zone_id := 0;
    L_History_Event.priority := E_ALERT_PRIORITY.ALERT_PRIORITY_HIGH;
    L_Last_Operator_Journal_Seq := GVL_STATUS.G_Diagnostics.Operator_Journal_Event_Seq;
END_IF;

// --- History anti-flood / dedup ---
IF L_History_Write_Event THEN
    IF (L_History_Event.event_code = L_Last_Event_Code)
       AND (ABS(L_History_Event.event_value - L_Last_Event_Value) < 0.001)
       AND (GVL_STATUS.G_System_Time_MS - L_Last_Event_Time_MS < 5000) THEN
        L_History_Write_Event := FALSE;
    ELSE
        L_Last_Event_Code := L_History_Event.event_code;
        L_Last_Event_Value := L_History_Event.event_value;
        L_Last_Event_Time_MS := GVL_STATUS.G_System_Time_MS;
    END_IF;
END_IF;

fbHistoryManager(
    VI_System_Time_MS := GVL_STATUS.G_System_Time_MS,
    VI_Write_Event := L_History_Write_Event,
    VI_Event := L_History_Event
);


L_Maintenance_Apply_Intent := FALSE;

// Dangerous action confirmation flow
IF GVL_COMMAND.CMD_Dangerous_Action_Request AND (GVL_COMMAND.CMD_User_Access_Level >= 2) THEN

    IF NOT L_Dangerous_Action_Armed THEN
        fbLogEvent(
            VI_Event_Type := 8,
            VI_Timestamp := GVL_STATUS.G_System_Time_MS,
            VI_Param1 := TO_UDINT(GVL_COMMAND.CMD_User_Access_Level),
            VI_Param2 := 1
        );
    END_IF;

    L_Dangerous_Action_Armed := TRUE;
    L_Dangerous_Action_Deadline_MS := GVL_STATUS.G_System_Time_MS + 15000;
    GVL_STATUS.G_Diagnostics.Dangerous_Action_Pending_Confirm := TRUE;
    GVL_STATUS.G_Diagnostics.Dangerous_Action_Confirm_Deadline_MS := L_Dangerous_Action_Deadline_MS;
    GVL_STATUS.G_Diagnostics.Dangerous_Action_Confirm_Text := 'Подтвердите опасное действие в течение 15 секунд';
END_IF;
IF L_Dangerous_Action_Armed AND (GVL_STATUS.G_System_Time_MS > L_Dangerous_Action_Deadline_MS) THEN
    L_Dangerous_Action_Armed := FALSE;
    GVL_STATUS.G_Diagnostics.Dangerous_Action_Pending_Confirm := FALSE;
    GVL_STATUS.G_Diagnostics.Dangerous_Action_Confirm_Text := 'Окно подтверждения истекло';
END_IF;
IF GVL_COMMAND.CMD_Dangerous_Action_Confirm AND
   L_Dangerous_Action_Armed AND
   (GVL_COMMAND.CMD_User_Access_Level >= 2) THEN
    L_Maintenance_Apply_Intent := TRUE;

    fbLogEvent(
        VI_Event_Type := 9,
        VI_Timestamp := GVL_STATUS.G_System_Time_MS,
        VI_Param1 := TO_UDINT(GVL_COMMAND.CMD_User_Access_Level),
        VI_Param2 := 1
    );

    L_Dangerous_Action_Armed := FALSE;
    GVL_STATUS.G_Diagnostics.Dangerous_Action_Pending_Confirm := FALSE;
    GVL_STATUS.G_Diagnostics.Dangerous_Action_Confirm_Text := 'Опасное действие подтверждено оператором';
END_IF;

// HMI maintenance mode control (confirmation-aware)
IF L_Maintenance_Apply_Intent THEN
    FOR L_i := 1 TO GVL_CONSTANTS.C_MAX_MANIFOLDS DO
        GVL_CONFIG.G_Manifold_Pump_In_Service[L_i] := GVL_COMMAND.CMD_Set_Manifold_Pump_In_Service[L_i];
    END_FOR;
    GVL_CONFIG.G_DHW_Heating_Pump_In_Service := GVL_COMMAND.CMD_Set_DHW_Heating_Pump_In_Service;
    GVL_CONFIG.G_DHW_Circ_Pump_In_Service := GVL_COMMAND.CMD_Set_DHW_Circ_Pump_In_Service;
END_IF;

// Access level enforcement for dangerous actions
GVL_STATUS.G_Diagnostics.User_Access_Level_Active := GVL_COMMAND.CMD_User_Access_Level;
GVL_STATUS.G_Diagnostics.User_Access_Denied := FALSE;
GVL_STATUS.G_Diagnostics.User_Access_Deny_Reason := '';
IF GVL_COMMAND.CMD_Dangerous_Action_Request OR GVL_COMMAND.CMD_Dangerous_Action_Confirm THEN
    IF GVL_COMMAND.CMD_User_Access_Level < 2 THEN
        IF NOT L_User_Access_Denied_Prev THEN
            fbLogEvent(
                VI_Event_Type := 10,
                VI_Timestamp := GVL_STATUS.G_System_Time_MS,
                VI_Param1 := TO_UDINT(GVL_COMMAND.CMD_User_Access_Level),
                VI_Param2 := 2
            );
        END_IF;

        GVL_STATUS.G_Diagnostics.User_Access_Denied := TRUE;
        GVL_STATUS.G_Diagnostics.User_Access_Deny_Reason := 'Недостаточный уровень доступа для опасного действия';
        GVL_STATUS.G_Diagnostics.Operator_Action_Blocked := TRUE;
        GVL_STATUS.G_Diagnostics.Operator_Block_Reason := 'Требуется уровень ENGINEER для опасного действия';
        GVL_STATUS.G_Diagnostics.Dangerous_Action_Pending_Confirm := FALSE;
        GVL_STATUS.G_Diagnostics.Dangerous_Action_Confirm_Text := 'Доступ запрещён: требуется уровень ENGINEER';
    END_IF;
END_IF;

L_User_Access_Denied_Prev := GVL_STATUS.G_Diagnostics.User_Access_Denied;

// Hard revert for forbidden operator actions
IF GVL_STATUS.G_Diagnostics.Operator_Action_Blocked THEN
    FOR L_i := 1 TO GVL_CONSTANTS.C_MAX_MANIFOLDS DO
        IF NOT GVL_CONFIG.G_Manifold_Pump_In_Service[L_i] THEN
            GVL_CONFIG.G_Manifold_Pump_In_Service[L_i] := TRUE;
        END_IF;
    END_FOR;
    IF NOT GVL_CONFIG.G_DHW_Heating_Pump_In_Service THEN
        GVL_CONFIG.G_DHW_Heating_Pump_In_Service := TRUE;
    END_IF;
    IF NOT GVL_CONFIG.G_DHW_Circ_Pump_In_Service THEN
        GVL_CONFIG.G_DHW_Circ_Pump_In_Service := TRUE;
    END_IF;
    GVL_STATUS.G_Diagnostics.Operator_Last_Forbidden_Action := GVL_STATUS.G_Diagnostics.Operator_Block_Reason;
END_IF;

